	  // nicht verwendete Signale für den 1. Schritt und eventuell weitere Schritte
	  (*#sxSendBuf.sxSTW1.Jog1         := False;
	          #sxSendBuf.sxSTW1.Jog2         := False;
	          #sxSendBuf.sxEPosSTW1.MdiTyp   := False;
	          #sxSendBuf.sxEPosSTW1.MdiPos   := False;
	          #sxSendBuf.sxEPosSTW1.MdiNeg   := False;
	          #sxSendBuf.sxEPosSTW1.MdiSetup := False;
	          #sxSendBuf.sxEPosSTW2.SetRefPt := False;
	          #sxSendBuf.sxEPosSTW2.JogInc   := False;
	          #sxSendBuf.sxEPosSTW2.RefStDi  := False;
	          #sxSendBuf.sxSTW1.RefStart     := False;
	          #sxSendBuf.sxEPosSTW2.RefTyp   := False;
	          #sxSendBuf.sxEPosSTW1.MdiStart := False;*)
	  #sxSendBuf.STW1.%X8 := False;
	  #sxSendBuf.STW1.%X9 := False;
	  #sxSendBuf.EPosSTW1.%X8 := False;
	  #sxSendBuf.EPosSTW1.%X9 := False;
	  #sxSendBuf.EPosSTW1.%X10 := False;
	  #sxSendBuf.EPosSTW1.%X14 := False;
	  #sxSendBuf.EPosSTW2.%X1 := False;
	  #sxSendBuf.EPosSTW2.%X5 := False;
	  #sxSendBuf.EPosSTW2.%X9 := False;
	  #sxSendBuf.STW1.%X11 := False;
	  #sxSendBuf.EPosSTW2.%X8 := False;
	  #sxSendBuf.EPosSTW1.%X15 := False;
	  
	  // Nach dem Einschalten des Antriebes, prüfen ob der Antrieb betriebsbereit, in Operation ohne Fehler und Warnung ist, 
	  // dann die Betriebsart MDI / Sollwertvorgabe Start gesetzt werden
	  IF #sbOff1 AND #sbReady AND #sbIOp AND NOT #sbFault THEN
	    
	    // Betriebsart MDI / Sollwertdirektvorgabe setzen
	    //#sxSendBuf.sxEPosSTW1.MdiStart := True;
	    #sxSendBuf.EPosSTW1.%X15 := True;
	    
	    // Positioniertyp auf absolutes Positionieren stellen 
	    //#sxSendBuf.sxEPosSTW1.MdiTyp := True;
	    #sxSendBuf.EPosSTW1.%X8 := True;
	    
	    // die Richtungswahl für das Positionieren auf positive Richtung oder negative Richtung einstellen
	    IF #Positive AND NOT #Negative THEN
	      
	      // positive Richtung
	      //#sxSendBuf.sxEPosSTW1.MdiPos := True;
	      #sxSendBuf.EPosSTW1.%X9 := True;
	      
	      // negative Richtung
	      //#sxSendBuf.sxEPosSTW1.MdiNeg := False;
	      #sxSendBuf.EPosSTW1.%X10 := False;
	      
	      // die Richtungswahl für das Positionieren auf negative Richtung einstellen                
	    ELSIF NOT #Positive AND #Negative THEN
	      
	      // positive Richtung
	      //#sxSendBuf.sxEPosSTW1.MdiPos := False;
	      #sxSendBuf.EPosSTW1.%X9 := False;
	      
	      // negative Richtung
	      //#sxSendBuf.sxEPosSTW1.MdiNeg := True;
	      #sxSendBuf.EPosSTW1.%X10 := True;
	      
	      // die Richtungswahl für das Positionieren auf keine Richtung einstellen                
	    ELSE
	      
	      // positive Richtung
	      //#sxSendBuf.sxEPosSTW1.MdiPos := False;
	      #sxSendBuf.EPosSTW1.%X9 := False;
	      
	      // negative Richtung
	      //#sxSendBuf.sxEPosSTW1.MdiNeg := False;
	      #sxSendBuf.EPosSTW1.%X10 := False;
	      
	    END_IF;
	    
	    // Nach dem Einschalten des Antriebes und dem Betriebsart MDI / Sollwertvorgabe starten, 
	    // ein Paar Zyklen warten bevor die Flanke für die Sollwertübernahme MDI gesetzt werden kann
	    IF #sbMdiStart AND (#siMdiStartCyc < #siCycWait) THEN
	      #siMdiStartCyc := #siMdiStartCyc + 1;
	    ELSE
	      // Flanke Sollwertübernahme MDI
	      //#sxSendBuf.sxSTW1.TrvStart := #Execute;
	      #sxSendBuf.STW1.%X6 := #sbExecute;
	      
	    END_IF;
	    
	    // "Fliegendes Referentieren" aktivieren
	    // "Fliegendes Referenzieren" erst nach Einschalten des Antriebes möglich
	    IF #sbRefTyp THEN
	      
	      // Referenziertyp auf "Fliegendes Referenzieren" einstellen
	      //#sxSendBuf.sxEPosSTW2.RefTyp := True;
	      #sxSendBuf.EPosSTW2.%X8 := True;
	      
	      // Nach der Anwahl des Referenziertyps "Fliegendes Referenzieren", 
	      // ein Zyklus später kann das Referenzieren gestartet
	      IF (#siRefTypCyc = 0) THEN
	        #siRefTypCyc := #siRefTypCyc + 1;
	      ELSE
	        // Referenzieren starten
	        //#sxSendBuf.sxSTW1.RefStart := True;
	        #sxSendBuf.STW1.%X11 := True;
	        
	      END_IF;
	    END_IF;
	  END_IF;
	  
	  // Betriebsart "Positionieren als Einrichten positiv" oder "Positionieren als Einrichten negativ"
	ELSIF #siModePos = 3 AND #sbModePos THEN
	  
	  // Antrieb einschalten
	  //#sxSendBuf.sxSTW1.Off1 := #sbOff1;
	  #sxSendBuf.STW1.%X0 := #sbOff1;
	  
	  // nicht verwendete Signale für den 1. Schritt und eventuell weitere Schritte
	  (*#sxSendBuf.sxSTW1.Jog1           := False;
	          #sxSendBuf.sxSTW1.Jog2           := False;
	          #sxSendBuf.sxEPosSTW1.MdiTyp     := False;
	          #sxSendBuf.sxEPosSTW1.MdiPos     := False;
	          #sxSendBuf.sxEPosSTW1.MdiNeg     := False;
	          #sxSendBuf.sxEPosSTW1.MdiSetup   := False;
	          #sxSendBuf.sxEPosSTW2.SetRefPt   := False;
	          #sxSendBuf.sxEPosSTW2.JogInc     := False;
	          #sxSendBuf.sxEPosSTW2.RefStDi    := False;
	          #sxSendBuf.sxSTW1.RefStart       := False;
	          #sxSendBuf.sxEPosSTW2.RefTyp     := False;
	          #sxSendBuf.sxEPosSTW1.MdiStart   := False;*)
	  #sxSendBuf.STW1.%X8 := False;
	  #sxSendBuf.STW1.%X9 := False;
	  #sxSendBuf.EPosSTW1.%X8 := False;
	  #sxSendBuf.EPosSTW1.%X9 := False;
	  #sxSendBuf.EPosSTW1.%X10 := False;
	  #sxSendBuf.EPosSTW1.%X14 := False;
	  #sxSendBuf.EPosSTW2.%X1 := False;
	  #sxSendBuf.EPosSTW2.%X5 := False;
	  #sxSendBuf.EPosSTW2.%X9 := False;
	  #sxSendBuf.STW1.%X11 := False;
	  #sxSendBuf.EPosSTW2.%X8 := False;
	  #sxSendBuf.EPosSTW1.%X15 := False;
	  
	  // Nach dem Einschalten des Antriebes, prüfen ob der Antrieb betriebsbereit, in Operation ohne Fehler und Warnung ist, 
	  // dann die Betriebsart MDI / Sollwertvorgabe Start gesetzt werden
	  IF #sbOff1 AND #sbReady AND #sbIOp AND NOT #sbFault THEN
	    
	    // Betriebsart MDI / Sollwertdirektvorgabe setzen
	    //#sxSendBuf.sxEPosSTW1.MdiStart := True;
	    #sxSendBuf.EPosSTW1.%X15 := True;
	    
	    // Positioniertyp auf absolutes Positionieren stellen 
	    //#sxSendBuf.sxEPosSTW1.MdiTyp := True;
	    #sxSendBuf.EPosSTW1.%X8 := True;
	    
	    // die Anwahl für MDI Modus auf Einrichten einstellen
	    //#sxSendBuf.sxEPosSTW1.MdiSetup := True;
	    #sxSendBuf.EPosSTW1.%X14 := True;
	    
	    // die Richtungswahl für das Positionieren auf positive Richtung oder negative Richtung einstellen
	    IF #Positive AND NOT #Negative THEN
	      
	      // positive Richtung
	      //#sxSendBuf.sxEPosSTW1.MdiPos := True;
	      #sxSendBuf.EPosSTW1.%X9 := True;
	      
	      // negative Richtung
	      //#sxSendBuf.sxEPosSTW1.MdiNeg := False;
	      #sxSendBuf.EPosSTW1.%X10 := False;
	      
	      // die Richtungswahl für das Positionieren auf negative Richtung einstellen                
	    ELSIF NOT #Positive AND #Negative THEN
	      
	      // positive Richtung
	      //#sxSendBuf.sxEPosSTW1.MdiPos := False;
	      #sxSendBuf.EPosSTW1.%X9 := False;
	      
	      // negative Richtung
	      //#sxSendBuf.sxEPosSTW1.MdiNeg := True;
	      #sxSendBuf.EPosSTW1.%X10 := True;
	      
	      // die Richtungswahl für das Positionieren auf keine Richtung einstellen                
	    ELSE
	      
	      // positive Richtung
	      //#sxSendBuf.sxEPosSTW1.MdiPos := False;
	      #sxSendBuf.EPosSTW1.%X9 := False;
	      
	      // negative Richtung
	      //#sxSendBuf.sxEPosSTW1.MdiNeg := False;
	      #sxSendBuf.EPosSTW1.%X10 := False;
	      
	    END_IF;
	    
	    // Nach dem Einschalten des Antriebes und dem Betriebsart MDI / Sollwertvorgabe starten, 
	    // ein Paar Zyklen warten bevor die Flanke für die Sollwertübernahme MDI gesetzt werden kann
	    IF #sbMdiStart AND (#siMdiStartCyc < #siCycWait) THEN
	      #siMdiStartCyc := #siMdiStartCyc + 1;
	    ELSE
	      // Flanke Sollwertübernahme MDI
	      //#sxSendBuf.sxSTW1.TrvStart := #Execute;
	      #sxSendBuf.STW1.%X6 := #sbExecute;
	      
	    END_IF;
	    
	    // "Fliegendes Referentieren" aktivieren
	    // "Fliegendes Referenzieren" erst nach Einschalten des Antriebes möglich
	    IF #sbRefTyp THEN
	      
	      // Referenziertyp auf "Fliegendes Referenzieren" einstellen
	      //#sxSendBuf.sxEPosSTW2.RefTyp := True;
	      #sxSendBuf.EPosSTW2.%X8 := True;
	      
	      // Nach der Anwahl des Referenziertyps "Fliegendes Referenzieren", 
	      // ein Zyklus später kann das Referenzieren gestartet
	      IF (#siRefTypCyc = 0) THEN
	        #siRefTypCyc := #siRefTypCyc + 1;
	      ELSE
	        // Referenzieren starten
	        //#sxSendBuf.sxSTW1.RefStart := True;
	        #sxSendBuf.STW1.%X11 := True;
	        
	      END_IF;
	    END_IF;
	  END_IF;
	  
	  // Hauptbetriebsart "Referenzieren" (Reference)
	  // Betriebsart "Referenzieren - Referenzpunktfahrt positiv" oder "Referenzieren - Referenzpunktfahrt negativ"
	ELSIF #siModePos = 4 AND #sbModePos THEN
	  
	  // Antrieb einschalten
	  //#sxSendBuf.sxSTW1.Off1 := #sbOff1;
	  #sxSendBuf.STW1.%X0 := #sbOff1;
	  
	  // nicht verwendete Signale für den 1. Schritt und eventuell weitere Schritte
	  (*#sxSendBuf.sxSTW1.Jog1         := False;
	          #sxSendBuf.sxSTW1.Jog2         := False;
	          #sxSendBuf.sxEPosSTW1.MdiStart := False;
	          #sxSendBuf.sxEPosSTW2.SetRefPt := False;
	          #sxSendBuf.sxEPosSTW2.JogInc   := False;
	          #sxSendBuf.sxEPosSTW2.RefTyp   := False;
	          #sxSendBuf.sxSTW1.RefStart     := False;
	          #sxSendBuf.sxEPosSTW2.RefStDi  := False;*)
	  #sxSendBuf.STW1.%X8 := False;
	  #sxSendBuf.STW1.%X9 := False;
	  #sxSendBuf.EPosSTW1.%X15 := False;
	  #sxSendBuf.EPosSTW2.%X1 := False;
	  #sxSendBuf.EPosSTW2.%X5 := False;
	  #sxSendBuf.EPosSTW2.%X8 := False;
	  #sxSendBuf.STW1.%X11 := False;
	  #sxSendBuf.EPosSTW2.%X9 := False;
	  
	  // Nach dem Einschalten des Antriebes, prüfen ob der Antrieb betriebsbereit, in Operation ohne Fehler und Warnung ist, 
	  // dann die Betriebsart MDI / Sollwertvorgabe Start gesetzt werden
	  IF #sbOff1 AND #sbReady AND #sbIOp AND NOT #sbFault THEN
	    
	    // Referenzieren starten
	    //#sxSendBuf.sxSTW1.RefStart := #Execute;
	    #sxSendBuf.STW1.%X11 := #sbExecute;
	    
	    // die Richtungswahl für das Referenzpunktfahrt positiv einstellen
	    IF #Positive AND NOT #Negative THEN
	      
	      // positive Referenzpunktfahrt
	      //#sxSendBuf.sxEPosSTW2.RefStDi := False;
	      #sxSendBuf.EPosSTW2.%X9 := False;
	      
	      // die Richtungswahl für das Referenzpunktfahrt negativ einstellen                
	    ELSIF NOT #Positive AND #Negative THEN
	      
	      // negative Referenzpunktfahrt
	      //#sxSendBuf.sxEPosSTW2.RefStDi := True;
	      #sxSendBuf.EPosSTW2.%X9 := True;
	      
	    END_IF;
	  END_IF;
	  
	  // Betriebsart "Referenzieren - Referenzpunkt setzen"
	ELSIF #siModePos = 5 AND #sbModePos THEN
	  
	  // Antrieb einschalten
	  //#sxSendBuf.sxSTW1.Off1 := #sbOff1;
	  #sxSendBuf.STW1.%X0 := #sbOff1;
	  
	  // nicht verwendete Signale für den 1. Schritt und eventuell weitere Schritte
	  (*#sxSendBuf.sxSTW1.Jog1          := False;
	          #sxSendBuf.sxSTW1.Jog2          := False;
	          #sxSendBuf.sxSTW1.RefStart      := False;
	          #sxSendBuf.sxEPosSTW1.MdiStart  := False;
	          #sxSendBuf.sxEPosSTW2.JogInc    := False;
	          #sxSendBuf.sxEPosSTW2.RefTyp    := False;
	          #sxSendBuf.sxEPosSTW2.RefStDi   := False;
	          #sxSendBuf.sxEPosSTW2.SetRefPt  := False;*)
	  #sxSendBuf.STW1.%X8 := False;
	  #sxSendBuf.STW1.%X9 := False;
	  #sxSendBuf.STW1.%X11 := False;
	  #sxSendBuf.EPosSTW1.%X15 := False;
	  #sxSendBuf.EPosSTW2.%X5 := False;
	  #sxSendBuf.EPosSTW2.%X8 := False;
	  #sxSendBuf.EPosSTW2.%X9 := False;
	  #sxSendBuf.EPosSTW2.%X1 := False;
	  
	  // Nach dem Einschalten des Antriebes, prüfen ob der Antrieb betriebsbereit, in Operation ohne Fehler und Warnung ist, 
	  // dann die Betriebsart MDI / Sollwertvorgabe Start gesetzt werden
	  IF NOT #sbFault THEN
	    
	    // Referenzpunktfahrt negativ
	    //#sxSendBuf.sxEPosSTW2.SetRefPt := #Execute;
	    #sxSendBuf.EPosSTW2.%X1 := #sbExecute;
	    
	  END_IF;
	  
	  // Hauptbetriebsart "Verfahrsätze" (Traversing Blocks)
	ELSIF #siModePos = 6 AND #sbModePos THEN
	  
	  // Antrieb einschalten
	  //#sxSendBuf.sxSTW1.Off1 := #sbOff1;
	  #sxSendBuf.STW1.%X0 := #sbOff1;
	  
	  // nicht verwendete Signale für den 1. Schritt und eventuell weitere Schritte
	  (*#sxSendBuf.sxSTW1.Jog1          := False;
	          #sxSendBuf.sxSTW1.Jog2          := False;
	          #sxSendBuf.sxEPosSTW1.MdiTyp    := False;
	          #sxSendBuf.sxEPosSTW1.MdiPos    := False;
	          #sxSendBuf.sxEPosSTW1.MdiNeg    := False;
	          #sxSendBuf.sxEPosSTW1.MdiSetup  := False;
	          #sxSendBuf.sxEPosSTW2.SetRefPt  := False;
	          #sxSendBuf.sxEPosSTW2.JogInc    := False;
	          #sxSendBuf.sxEPosSTW2.RefStDi   := False;
	          #sxSendBuf.sxEPosSTW2.RefTyp    := False;
	          #sxSendBuf.sxSTW1.RefStart      := False;
	          #sxSendBuf.sxEPosSTW1.TrvBit0   := False;
	          #sxSendBuf.sxEPosSTW1.TrvBit1   := False;
	          #sxSendBuf.sxEPosSTW1.TrvBit2   := False;
	          #sxSendBuf.sxEPosSTW1.TrvBit3   := False;
	          #sxSendBuf.sxEPosSTW1.TrvBit4   := False;
	          #sxSendBuf.sxEPosSTW1.TrvBit5   := False;
	          #sxSendBuf.sxEPosSTW1.MdiStart  := False;*)
	  #sxSendBuf.STW1.%X8 := False;
	  #sxSendBuf.STW1.%X9 := False;
	  #sxSendBuf.EPosSTW1.%X8 := False;
	  #sxSendBuf.EPosSTW1.%X9 := False;
	  #sxSendBuf.EPosSTW1.%X10 := False;
	  #sxSendBuf.EPosSTW1.%X14 := False;
	  #sxSendBuf.EPosSTW2.%X1 := False;
	  #sxSendBuf.EPosSTW2.%X5 := False;
	  #sxSendBuf.EPosSTW2.%X9 := False;
	  #sxSendBuf.EPosSTW2.%X8 := False;
	  #sxSendBuf.STW1.%X11 := False;
	  #sxSendBuf.EPosSTW1.%X0 := False;
	  #sxSendBuf.EPosSTW1.%X1 := False;
	  #sxSendBuf.EPosSTW1.%X2 := False;
	  #sxSendBuf.EPosSTW1.%X3 := False;
	  #sxSendBuf.EPosSTW1.%X4 := False;
	  #sxSendBuf.EPosSTW1.%X5 := False;
	  #sxSendBuf.EPosSTW1.%X15 := False;
	  
	  // Bei der Auswahl der Verfahrsätze entspricht die Position der Verfahrensatznummer 
	  // Verfahrsatznummer aus der Position ermitteln und in die einzelnen Bit's aufteilen
	  // Es sind die Verfahrsatznummern 0 - 63 möglich
	  IF (DINT_TO_INT(#Position) < 0) OR (DINT_TO_INT(#Position) > 63) THEN
	    // Fehler, ungültiger Verfahrsatznummer
	    #swStatus := 16#8204;
	    #Error := True;
	  ELSE
	    // Fehler wieder zurücknehmen, wenn er mal ausgelöst wurde
	    IF #swStatus = 16#8204 THEN
	      #swStatus := 16#7002;
	      #Error := False;
	    END_IF;
	    
	    // Verfahrsatznummer Bit 0 ermitteln
	    IF (DINT_TO_WORD(#Position) AND W#16#01) = W#16#01 THEN
	      //#sxSendBuf.sxEPosSTW1.TrvBit0 := True;
	      #sxSendBuf.EPosSTW1.%X0 := True;
	    END_IF;
	    
	    // Verfahrsatznummer Bit 1 ermitteln
	    IF (DINT_TO_WORD(#Position) AND W#16#02) = W#16#02 THEN
	      //#sxSendBuf.sxEPosSTW1.TrvBit1 := True;
	      #sxSendBuf.EPosSTW1.%X1 := True;
	    END_IF;
	    
	    // Verfahrsatznummer Bit 2 ermitteln
	    IF (DINT_TO_WORD(#Position) AND W#16#04) = W#16#04 THEN
	      //#sxSendBuf.sxEPosSTW1.TrvBit2 := True;
	      #sxSendBuf.EPosSTW1.%X2 := True;
	    END_IF;
	    
	    // Verfahrsatznummer Bit 3 ermitteln
	    IF (DINT_TO_WORD(#Position) AND W#16#08) = W#16#08 THEN
	      //#sxSendBuf.sxEPosSTW1.TrvBit3 := True;
	      #sxSendBuf.EPosSTW1.%X3 := True;
	    END_IF;
	    
	    // Verfahrsatznummer Bit 4 ermitteln
	    IF (DINT_TO_WORD(#Position) AND W#16#10) = W#16#10 THEN
	      //#sxSendBuf.sxEPosSTW1.TrvBit4 := True;
	      #sxSendBuf.EPosSTW1.%X4 := True;
	    END_IF;
	    
	    // Verfahrsatznummer Bit 5 ermitteln
	    IF (DINT_TO_WORD(#Position) AND W#16#20) = W#16#20 THEN
	      //#sxSendBuf.sxEPosSTW1.TrvBit5 := True;
	      #sxSendBuf.EPosSTW1.%X5 := True;
	    END_IF;
	    
	    // Nach dem Einschalten des Antriebes, prüfen ob der Antrieb betriebsbereit, in Operation ohne Fehler und Warnung ist, 
	    // dann die Betriebsart MDI / Sollwertvorgabe Start gesetzt werden
	    IF #sbOff1 AND #sbReady AND #sbIOp AND NOT #sbFault THEN
	      
	      #sxSendBuf.STW1.%X6 := #sbExecute;
	      
	      // "Fliegendes Referentieren" aktivieren
	      // "Fliegendes Referenzieren" erst nach Einschalten des Antriebes möglich
	      IF #sbRefTyp THEN
	        
	        // Referenziertyp auf "Fliegendes Referenzieren" einstellen
	        //#sxSendBuf.sxEPosSTW2.RefTyp := True;
	        #sxSendBuf.EPosSTW2.%X8 := True;
	        
	        // Nach der Anwahl des Referenziertyps "Fliegendes Referenzieren", 
	        // ein Zyklus später kann das Referenzieren gestartet
	        IF (#siRefTypCyc = 0) THEN
	          #siRefTypCyc := #siRefTypCyc + 1;
	        ELSE
	          // Referenzieren starten
	          //#sxSendBuf.sxSTW1.RefStart := True;
	          #sxSendBuf.STW1.%X11 := True;
	        END_IF;
	      END_IF;
	    END_IF;
	  END_IF;
	  
	  // Hauptbetriebsart "Tippen" (Jogging)
	  // Betriebsart "Tippen positiv" oder "Tippen negativ" angewählt 
	ELSIF #siModePos = 7 AND #sbModePos THEN
	  
	  // Antrieb einschalten
	  //#sxSendBuf.sxSTW1.Off1 := #sbOff1;
	  #sxSendBuf.STW1.%X0 := #sbOff1;
	  
	  // nicht verwendete Signale für den 1. Schritt und eventuell weitere Schritte
	  (*#sxSendBuf.sxEPosSTW1.MdiStart := False;
	          #sxSendBuf.sxEPosSTW2.JogInc   := False;
	          #sxSendBuf.sxSTW1.Jog1         := False;
	          #sxSendBuf.sxSTW1.Jog2         := False;
	          #sxSendBuf.sxEPosSTW2.RefTyp   := False;
	          #sxSendBuf.sxSTW1.RefStart     := False;
	          #sxSendBuf.sxEPosSTW2.SetRefPt  := False;*)
	  
	  #sxSendBuf.EPosSTW1.%X15 := False;
	  #sxSendBuf.EPosSTW2.%X5 := False;
	  #sxSendBuf.STW1.%X8 := False;
	  #sxSendBuf.STW1.%X9 := False;
	  #sxSendBuf.EPosSTW2.%X8 := False;
	  #sxSendBuf.STW1.%X11 := False;
	  #sxSendBuf.EPosSTW2.%X1 := False;
	  
	  // Nach dem Einschalten des Antriebes, prüfen ob der Antrieb betriebsbereit, in Operation ohne Fehler und Warnung ist, 
	  // dann kann Tippen positiv oder negativ gesetzt werden
	  IF #sbOff1 AND #sbReady AND #sbIOp AND NOT #sbFault THEN
	    
	    // Tippen positiv
	    IF #Jog1 AND NOT #Jog2 THEN
	      //#sxSendBuf.sxSTW1.Jog1 := True;
	      #sxSendBuf.STW1.%X8 := True;
	    END_IF;
	    
	    // Tippen negativ
	    IF #Jog2 AND NOT #Jog1 THEN
	      //#sxSendBuf.sxSTW1.Jog2 := True;
	      #sxSendBuf.STW1.%X9 := True;
	    END_IF;
	    
	    // "Fliegendes Referentieren" aktivieren
	    // "Fliegendes Referenzieren" erst nach Einschalten des Antriebes möglich
	    IF #sbRefTyp THEN
	      
	      // Referenziertyp auf "Fliegendes Referenzieren" einstellen
	      //#sxSendBuf.sxEPosSTW2.RefTyp := #FlyRef;
	      #sxSendBuf.EPosSTW2.%X8 := #FlyRef;
	      
	      // Nach der Anwahl des Referenziertyps "Fliegendes Referenzieren", 
	      // ein Zyklus später kann das Referenzieren gestartet
	      IF (#siRefTypCyc = 0) THEN
	        #siRefTypCyc := #siRefTypCyc + 1;
	      ELSE
	        // Referenzieren starten
	        //#sxSendBuf.sxSTW1.RefStart := True;
	        #sxSendBuf.STW1.%X11 := True;
	      END_IF;
	    END_IF;
	  END_IF;
	  
	  // Betriebsart "Tippen positiv / Tippen negativ inkrementell" 
	ELSIF #siModePos = 8 AND #sbModePos THEN
	  
	  // Antrieb einschalten
	  //#sxSendBuf.sxSTW1.OFF1 := #sbOff1;
	  #sxSendBuf.STW1.%X0 := #sbOff1;
	  
	  // nicht verwendete Signale für den 1. Schritt und eventuell weitere Schritte
	  (*#sxSendBuf.sxEPosSTW1.MdiStart := False;
	          #sxSendBuf.sxEPosSTW2.JogInc   := False;
	          #sxSendBuf.sxSTW1.Jog1         := False;
	          #sxSendBuf.sxSTW1.Jog2         := False;
	          #sxSendBuf.sxSTW1.RefStart     := False;
	          #sxSendBuf.sxEPosSTW2.RefTyp   := False;
	          #sxSendBuf.sxEPosSTW2.SetRefPt  := False;*)
	  
	  #sxSendBuf.EPosSTW1.%X15 := False;
	  #sxSendBuf.EPosSTW2.%X5 := False;
	  #sxSendBuf.STW1.%X8 := False;
	  #sxSendBuf.STW1.%X9 := False;
	  #sxSendBuf.STW1.%X11 := False;
	  #sxSendBuf.EPosSTW2.%X8 := False;
	  #sxSendBuf.EPosSTW2.%X1 := False;
	  
	  // Nach dem Einschalten des Antriebes, ein Paar Zyklen warten bevor Tippen negativ gesetzt werden kann
	  // Nach dem Einschalten des Antriebes, prüfen ob der Antrieb betriebsbereit, in Operation ohne Fehler und Warnung ist, 
	  // dann kann Tippen positiv oder negativ gesetzt werden
	  IF #sbOff1 AND #sbReady AND #sbIOp AND NOT #sbFault THEN
	    
	    // Tippen inkrementell einstellen
	    //#sxSendBuf.sxEPosSTW2.JogInc := True;
	    #sxSendBuf.EPosSTW2.%X5 := True;
	    
	    #sbJogInc := True;
	    
	    // Nach dem Einstellen des Antriebes, ein Paar Zyklen warten bevor Tippen negativ oder Tippen positiv gesetz werden kann
	    IF #sbJogInc AND (#siJogIncCyc = 0) THEN
	      #siJogIncCyc := #siJogIncCyc + 1;
	    ELSE
	      
	      // Tippen positiv oder negativ inkrementell zulassen
	      IF #Jog1 XOR #Jog2 THEN
	        
	        //#sxSendBuf.sxSTW1.Jog1 := #Jog1;
	        //#sxSendBuf.sxSTW1.Jog2 := #Jog2;
	        #sxSendBuf.STW1.%X8 := #Jog1;
	        #sxSendBuf.STW1.%X9 := #Jog2;
	      END_IF;
	    END_IF;
	    
	    // "Fliegendes Referentieren" aktivieren
	    // "Fliegendes Referenzieren" erst nach Einschalten des Antriebes möglich
	    IF #sbRefTyp THEN
	      
	      // Referenziertyp auf "Fliegendes Referenzieren" einstellen
	      //#sxSendBuf.sxEPosSTW2.RefTyp := True;
	      #sxSendBuf.EPosSTW2.%X8 := True;
	      
	      // Nach der Anwahl des Referenziertyps "Fliegendes Referenzieren", 
	      // ein Zyklus später kann das Referenzieren gestartet
	      IF (#siRefTypCyc = 0) THEN
	        #siRefTypCyc := #siRefTypCyc + 1;
	      ELSE
	        // Referenzieren starten
	        //#sxSendBuf.sxSTW1.RefStart := True;
	        #sxSendBuf.STW1.%X11 := True;
	      END_IF;
	    END_IF;
	  END_IF;
	ELSE
	  // Werte wieder zurücknehmen
	  (*#sxSendBuf.sxSTW1.Off1          := #Off1;
	          #sxSendBuf.sxSTW1.RejTrvTsk     := False;
	          #sxSendBuf.sxSTW1.TrvStart      := False;
	          #sxSendBuf.sxEPosSTW1.MdiStart  := False;
	          #sxSendBuf.sxSTW1.Jog1          := False;
	          #sxSendBuf.sxSTW1.Jog2          := False;
	          #sxSendBuf.sxEPosSTW1.MdiTyp    := False;
	          #sxSendBuf.sxEPosSTW1.MdiPos    := False;
	          #sxSendBuf.sxEPosSTW1.MdiNeg    := False;
	          #sxSendBuf.sxEPosSTW1.MdiTrTyp  := False;
	          #sxSendBuf.sxEPosSTW1.MdiSetup  := False;
	          #sxSendBuf.sxEPosSTW2.SetRefPt  := False;
	          #sxSendBuf.sxEPosSTW2.RefTyp    := False;
	          #sxSendBuf.sxEPosSTW2.RefStDi   := False;
	          #sxSendBuf.sxEPosSTW2.JogInc    := False;
	          #sxSendBuf.sxSTW1.RefStart      := False;*)
	  
	  #sxSendBuf.STW1.%X0 := #EnableAxis;
	  #sxSendBuf.STW1.%X4 := False;
	  #sxSendBuf.STW1.%X6 := False;
	  #sxSendBuf.EPosSTW1.%X15 := False;
	  #sxSendBuf.STW1.%X8 := False;
	  #sxSendBuf.STW1.%X9 := False;
	  #sxSendBuf.EPosSTW1.%X8 := False;
	  #sxSendBuf.EPosSTW1.%X9 := False;
	  #sxSendBuf.EPosSTW1.%X10 := False;
	  #sxSendBuf.EPosSTW1.%X12 := False;
	  #sxSendBuf.EPosSTW1.%X14 := False;
	  #sxSendBuf.EPosSTW2.%X1 := False;
	  #sxSendBuf.EPosSTW2.%X8 := False;
	  #sxSendBuf.EPosSTW2.%X9 := False;
	  #sxSendBuf.EPosSTW2.%X5 := False;
	  #sxSendBuf.STW1.%X11 := False;
	END_IF; // Hauptbetriebsart "Verfahrsätze" (Traversing Blocks)
	
	//Den Eingang ConfigEPos auf die einzelnen Bits im Telegramm verschalten
	#sxSendBuf.STW1.%X1 := #ConfigEPos.%X0;
	#sxSendBuf.STW1.%X2 := #ConfigEPos.%X1;
	#sxSendBuf.EPosSTW2.%X14 := #ConfigEPos.%X2;
	#sxSendBuf.EPosSTW2.%X15 := #ConfigEPos.%X3;
	#sxSendBuf.EPosSTW2.%X11 := #ConfigEPos.%X4;
	#sxSendBuf.EPosSTW2.%X10 := #ConfigEPos.%X5;
	#sxSendBuf.EPosSTW2.%X2 := #ConfigEPos.%X6;
	#sxSendBuf.STW1.%X13 := #ConfigEPos.%X7;
	#sxSendBuf.EPosSTW1.%X12 := #ConfigEPos.%X8;
	#sxSendBuf.STW2.%X0 := #ConfigEPos.%X9;
	#sxSendBuf.STW2.%X1 := #ConfigEPos.%X10;
	#sxSendBuf.STW2.%X2 := #ConfigEPos.%X11;
	#sxSendBuf.STW2.%X3 := #ConfigEPos.%X12;
	#sxSendBuf.STW2.%X4 := #ConfigEPos.%X13;
	#sxSendBuf.STW2.%X7 := #ConfigEPos.%X14;
	#sxSendBuf.STW1.%X12 := #ConfigEPos.%X15;
	#sxSendBuf.STW1.%X14 := #ConfigEPos.%X16;
	#sxSendBuf.STW1.%X15 := #ConfigEPos.%X17;
	#sxSendBuf.EPosSTW1.%X6 := #ConfigEPos.%X18;
	#sxSendBuf.EPosSTW1.%X7 := #ConfigEPos.%X19;
	#sxSendBuf.EPosSTW1.%X11 := #ConfigEPos.%X20;
	#sxSendBuf.EPosSTW1.%X13 := #ConfigEPos.%X21;
	#sxSendBuf.EPosSTW2.%X3 := #ConfigEPos.%X22;
	#sxSendBuf.EPosSTW2.%X4 := #ConfigEPos.%X23;
	#sxSendBuf.EPosSTW2.%X6 := #ConfigEPos.%X24;
	#sxSendBuf.EPosSTW2.%X7 := #ConfigEPos.%X25;
	#sxSendBuf.EPosSTW2.%X12 := #ConfigEPos.%X26;
	#sxSendBuf.EPosSTW2.%X13 := #ConfigEPos.%X27;
	#sxSendBuf.STW2.%X5 := #ConfigEPos.%X28;
	#sxSendBuf.STW2.%X6 := #ConfigEPos.%X29;
	#sxSendBuf.STW2.%X8 := #ConfigEPos.%X30;
	#sxSendBuf.STW2.%X9 := #ConfigEPos.%X31;
	
	
	#swSendBuf[0] := #sxSendBuf.STW1;
	#swSendBuf[1] := #sxSendBuf.EPosSTW1;
	#swSendBuf[2] := #sxSendBuf.EPosSTW2;
	#swSendBuf[3] := #sxSendBuf.STW2;
	#swSendBuf[4] := #sxSendBuf.OverrideV;
	#swSendBuf[5] := #sxSendBuf.Position.%W1;
	#swSendBuf[6] := #sxSendBuf.Position.%W0;
	#swSendBuf[7] := #sxSendBuf.Velocity.%W1;
	#swSendBuf[8] := #sxSendBuf.Velocity.%W0;
	#swSendBuf[9] := #sxSendBuf.OverrideA;
	#swSendBuf[10] := #sxSendBuf.OverrideD;
	#swSendBuf[11] := #sxSendBuf.Reserve;
	
	//Prozessdaten zur Signalbaugruppe schreiben
	#piRetSFC := DPWR_DAT(LADDR := #HWIDSTW,
	                      RECORD := #swSendBuf);
	
	// Fehler der Rückmeldung ausgeben
	#DiagID := INT_TO_WORD(#piRetSFC);
	
	//kein Fehler beim Schreiben
	IF #piRetSFC = 0 THEN
	  
	  // Fehler wieder zurück nehmen
	  IF (#swStatus = 16#8601) THEN
	    #swStatus := 16#7002;
	    #Error := False;
	  END_IF;
	  
	  //Prozessdaten von der Signalbaugruppe lesen
	  #piRetSFC := DPRD_DAT(LADDR := #HWIDZSW,
	                        RECORD => #swRecvBuf);
	  
	  // Fehlermeldung der Rückmeldung ausgeben
	  #DiagID := INT_TO_WORD(#piRetSFC);
	  
	  //Fehler beim Lesen (Profibus-Kommunikation unterbrochen)
	  IF #piRetSFC <> 0 THEN
	    
	    // Fehler
	    #Error := TRUE;
	    #swStatus := 16#8600;
	    
	    // Zustandsworte löschen
	    #sxRecvBuf.ZSW1 := W#16#0;
	    #sxRecvBuf.EPosZSW1 := W#16#0;
	    #sxRecvBuf.EPosZSW2 := W#16#0;
	    #sxRecvBuf.ZSW2 := W#16#0;
	    #sxRecvBuf.NotUsed := W#16#00;
	    #sxRecvBuf.Position := DW#16#00;
	    #sxRecvBuf.Velocity := DW#16#00;
	    #sxRecvBuf.ErrNr := W#16#00;
	    #sxRecvBuf.WarnNr := W#16#00;
	    #sxRecvBuf.Reserve := W#16#00;
	    
	    // Werte auslesen
	  ELSE
	    
	    // Fehler wieder zurück nehmen
	    IF (#swStatus = 16#8600) THEN
	      #swStatus := 16#7002;
	      #Error := False;
	    END_IF;
	    
	    #sxRecvBuf.ZSW1 := #swRecvBuf[0];
	    #sxRecvBuf.EPosZSW1 := #swRecvBuf[1];
	    #sxRecvBuf.EPosZSW2 := #swRecvBuf[2];
	    #sxRecvBuf.ZSW2 := #swRecvBuf[3];
	    #sxRecvBuf.NotUsed := #swRecvBuf[4];
	    #sxRecvBuf.Position.%W1 := #swRecvBuf[5];
	    #sxRecvBuf.Position.%W0 := #swRecvBuf[6];
	    #sxRecvBuf.Velocity.%W1 := #swRecvBuf[7];
	    #sxRecvBuf.Velocity.%W0 := #swRecvBuf[8];
	    #sxRecvBuf.ErrNr := #swRecvBuf[9];
	    #sxRecvBuf.WarnNr := #swRecvBuf[10];
	    #sxRecvBuf.Reserve := #swRecvBuf[11];
	    
	    // ZSW1 aufbereiten
	    //#Busy := #sxRecvBuf.sxZSW1.IOp;
	    #sbBusy := #sxRecvBuf.ZSW1.%X2;
	    
	    // Fehler auswerten
	    IF #sxRecvBuf.ZSW1.%X3 THEN
	      #swStatus := 16#8401;
	      #Error := True;
	    ELSIF #sxRecvBuf.ZSW1.%X6 THEN
	      #swStatus := 16#8402;
	      #Error := True;
	    ELSE
	      // Fehler wieder zurück nehmen
	      IF (#swStatus = 16#8401) OR (#swStatus = 16#8402) THEN
	        #swStatus := 16#7002;
	        #Error := False;
	      END_IF;
	    END_IF;
	    
	    // EPOS_ZSW1            
	    // EPOS-Wort-1 BIT 00 --> 1 = Active traversing block bit 0
	    //IF #sxRecvBuf.sxEPosZSW1.ActTrvBit0 THEN
	    IF #sxRecvBuf.EPosZSW1.%X0 THEN
	      #swEPosZSW1 := #swEPosZSW1 OR W#16#01;
	    ELSE
	      #swEPosZSW1 := #swEPosZSW1 AND W#16#FFFE;
	    END_IF;
	    
	    // EPOS-Wort-1 Bit 01 --> 1 = Active traversing block bit 1
	    //IF #sxRecvBuf.sxEPosZSW1.ActTrvBit1 THEN
	    IF #sxRecvBuf.EPosZSW1.%X1 THEN
	      #swEPosZSW1 := #swEPosZSW1 OR W#16#02;
	    ELSE
	      #swEPosZSW1 := #swEPosZSW1 AND W#16#FFFD;
	    END_IF;
	    
	    // EPOS-Wort-1 Bit 02 --> 1 = Active traversing block bit 2
	    //IF #sxRecvBuf.sxEPosZSW1.ActTrvBit2 THEN
	    IF #sxRecvBuf.EPosZSW1.%X2 THEN
	      #swEPosZSW1 := #swEPosZSW1 OR W#16#04;
	    ELSE
	      #swEPosZSW1 := #swEPosZSW1 AND W#16#FFFB;
	    END_IF;
	    
	    // EPOS-Wort-1 Bit 03 --> 1 = Active traversing block bit 3
	    //IF #sxRecvBuf.sxEPosZSW1.ActTrvBit3 THEN
	    IF #sxRecvBuf.EPosZSW1.%X3 THEN
	      #swEPosZSW1 := #swEPosZSW1 OR W#16#08;
	    ELSE
	      #swEPosZSW1 := #swEPosZSW1 AND W#16#FFF7;
	    END_IF;
	    
	    // EPOS-Wort-1 Bit 04 --> 1 = Active traversing block bit 4 
	    //IF #sxRecvBuf.sxEPosZSW1.ActTrvBit4 THEN
	    IF #sxRecvBuf.EPosZSW1.%X4 THEN
	      #swEPosZSW1 := #swEPosZSW1 OR W#16#10;
	    ELSE
	      #swEPosZSW1 := #swEPosZSW1 AND W#16#FFEF;
	    END_IF;
	    
	    // EPOS-Wort-1 Bit 05 --> 1 = Active traversing block bit 5
	    //IF #sxRecvBuf.sxEPosZSW1.ActTrvBit5 THEN
	    IF #sxRecvBuf.EPosZSW1.%X5 THEN
	      #swEPosZSW1 := #swEPosZSW1 OR W#16#20;
	    ELSE
	      #swEPosZSW1 := #swEPosZSW1 AND W#16#FFDF;
	    END_IF;
	    
	    // EPOS-Wort-1 Bit 08 --> 1 = STOP cam minus active
	    //IF #sxRecvBuf.sxEPosZSW1.StpCamMinAct THEN
	    IF #sxRecvBuf.EPosZSW1.%X8 THEN
	      #swEPosZSW1 := #swEPosZSW1 OR W#16#100;
	    ELSE
	      #swEPosZSW1 := #swEPosZSW1 AND W#16#FEFF;
	    END_IF;
	    
	    // EPOS-Wort-1 Bit 09 --> 1 = STOP cam plus active
	    //IF #sxRecvBuf.sxEPosZSW1.StpCamPlsAct THEN
	    IF #sxRecvBuf.EPosZSW1.%X9 THEN
	      #swEPosZSW1 := #swEPosZSW1 OR W#16#200;
	    ELSE
	      #swEPosZSW1 := #swEPosZSW1 AND W#16#FDFF;
	    END_IF;
	    
	    // EPOS-Wort-1 Bit 10 --> 1 = Jogging active
	    //IF #sxRecvBuf.sxEPosZSW1.JogAct THEN
	    IF #sxRecvBuf.EPosZSW1.%X10 THEN
	      #swEPosZSW1 := #swEPosZSW1 OR W#16#400;
	    ELSE
	      #swEPosZSW1 := #swEPosZSW1 AND W#16#FBFF;
	    END_IF;
	    
	    // EPOS-Wort-1 Bit 11 --> 1 = Reference point approach active
	    //IF #sxRecvBuf.sxEPosZSW1.RefAct THEN
	    IF #sxRecvBuf.EPosZSW1.%X11 THEN
	      #swEPosZSW1 := #swEPosZSW1 OR W#16#800;
	    ELSE
	      #swEPosZSW1 := #swEPosZSW1 AND W#16#F7FF;
	    END_IF;
	    
	    // Anstossen des fliegenden Referenzieren prüfen, wenn die Rückmeldung fehlt dann wiederholen
	    //IF NOT #sxRecvBuf.sxEPosZSW1.FlyRefAct AND #sbRefTyp AND #sxSendBuf.sxSTW1.RefStart THEN
	    IF NOT #sxRecvBuf.EPosZSW1.%X12 AND #sbRefTyp AND #sxSendBuf.STW1.%X11 THEN
	      
	      // Wiederholung anstossen 
	      IF #siRefActRetry < #siRetryMax THEN
	        #siRefActRetry := #siRefActRetry + 1;
	        
	        // Referenzieren starten wieder wegnehmen
	        //#sxSendBuf.sxSTW1.RefStart := False;
	        #sxSendBuf.STW1.%X11 := False;
	      ELSE
	        
	        // Fehlermeldung
	        #swStatus := 16#8403;
	        #Error := True;
	      END_IF;
	    ELSE
	      
	      // Fehler wieder zurücknehmen, wenn er mal ausgelöst wurde
	      IF #swStatus = 16#8403 THEN
	        #swStatus := 16#7002;
	        #Error := False;
	      END_IF;
	      // Zähler zurücksetzen bei Rückmeldung fliegendes Referenzieren jetzt aktiviert oder bei Abwahl der Funktion
	      IF (#sxRecvBuf.EPosZSW1.%X12 AND #sbRefTyp AND #sxSendBuf.STW1.%X11) OR NOT #FlyRef THEN
	        #siRefActRetry := 0;
	      END_IF;
	    END_IF;
	    
	    // EPOS-Wort-1 Bit 12 --> 1 = Flying referencing active
	    //IF #sxRecvBuf.sxEPosZSW1.FlyRefAct THEN
	    IF #sxRecvBuf.EPosZSW1.%X12 THEN
	      #swEPosZSW1 := #swEPosZSW1 OR W#16#1000;
	    ELSE
	      #swEPosZSW1 := #swEPosZSW1 AND W#16#EFFF;
	    END_IF;
	    
	    // EPOS-Wort-1 Bit 13 --> 1 = Traversing block active
	    //IF #sxRecvBuf.sxEPosZSW1.TrvBlAct THEN
	    IF #sxRecvBuf.EPosZSW1.%X13 THEN
	      #swEPosZSW1 := #swEPosZSW1 OR W#16#2000;
	    ELSE
	      #swEPosZSW1 := #swEPosZSW1 AND W#16#DFFF;
	    END_IF;
	    
	    // EPOS-Wort-1 Bit 14 --> 1 = MDI setup active
	    //IF #sxRecvBuf.sxEPosZSW1.MdiStupAct THEN
	    IF #sxRecvBuf.EPosZSW1.%X14 THEN
	      #swEPosZSW1 := #swEPosZSW1 OR W#16#4000;
	    ELSE
	      #swEPosZSW1 := #swEPosZSW1 AND W#16#BFFF;
	    END_IF;
	    
	    // EPOS-Wort-1 Bit 15 --> 1 = MDI positing active
	    //IF #sxRecvBuf.sxEPosZSW1.MdiPosAct THEN
	    IF #sxRecvBuf.EPosZSW1.%X15 THEN
	      #swEPosZSW1 := #swEPosZSW1 OR W#16#8000;
	    ELSE
	      #swEPosZSW1 := #swEPosZSW1 AND W#16#7FFF;
	    END_IF;
	    
	    // EPOS_ZSW2 
	    // EPOS-Wort-2 Bit 00 --> 1 = Tracking mode active
	    //IF #sxRecvBuf.sxEPosZSW2.TrkModeAct THEN
	    IF #sxRecvBuf.EPosZSW2.%X0 THEN
	      #swEPosZSW2 := #swEPosZSW2 OR W#16#01;
	    ELSE
	      #swEPosZSW2 := #swEPosZSW2 AND W#16#FFFE;
	    END_IF;
	    
	    // EPOS-Wort-2 Bit 01 --> 1 = Velocity limit active
	    //IF #sxRecvBuf.sxEPosZSW2.VeloLimAct THEN
	    IF #sxRecvBuf.EPosZSW2.%X1 THEN
	      #swEPosZSW2 := #swEPosZSW2 OR W#16#02;
	    ELSE
	      #swEPosZSW2 := #swEPosZSW2 AND W#16#FFFD;
	    END_IF;
	    
	    // EPOS-Wort-2 Bit 02 --> 1 = Setpoint static
	    //IF #sxRecvBuf.sxEPosZSW2.SetPStat THEN
	    IF #sxRecvBuf.EPosZSW2.%X2 THEN
	      #swEPosZSW2 := #swEPosZSW2 OR W#16#04;
	    ELSE
	      #swEPosZSW2 := #swEPosZSW2 AND W#16#FFFB;
	    END_IF;
	    
	    // EPOS-Wort-2 Bit 03 --> 1 = Printmark outside outer window
	    //IF #sxRecvBuf.sxEPosZSW2.PrnMrkOut THEN
	    IF #sxRecvBuf.EPosZSW2.%X3 THEN
	      #swEPosZSW2 := #swEPosZSW2 OR W#16#08;
	    ELSE
	      #swEPosZSW2 := #swEPosZSW2 AND W#16#FFF7;
	    END_IF;
	    
	    // EPOS-Wort-2 Bit 04 --> 1 = Axis forwards
	    //IF #sxRecvBuf.sxEPosZSW2.FWD THEN
	    IF #sxRecvBuf.EPosZSW2.%X4 THEN
	      #swEPosZSW2 := #swEPosZSW2 OR W#16#10;
	    ELSE
	      #swEPosZSW2 := #swEPosZSW2 AND W#16#FFEF;
	    END_IF;
	    
	    // EPOS-Wort-2 Bit 05 --> 1 = Axis backwards
	    //IF #sxRecvBuf.sxEPosZSW2.BWD THEN
	    IF #sxRecvBuf.EPosZSW2.%X5 THEN
	      #swEPosZSW2 := #swEPosZSW2 OR W#16#20;
	    ELSE
	      #swEPosZSW2 := #swEPosZSW2 AND W#16#FFDF;
	    END_IF;
	    
	    // EPOS-Wort-2 Bit 06 --> 1 = Software limit switch minus active
	    //IF #sxRecvBuf.sxEPosZSW2.SftSwMinAct THEN
	    IF #sxRecvBuf.EPosZSW2.%X6 THEN
	      #swEPosZSW2 := #swEPosZSW2 OR W#16#40;
	    ELSE
	      #swEPosZSW2 := #swEPosZSW2 AND W#16#FFBF;
	    END_IF;
	    
	    // EPOS-Wort-2 Bit 07 --> 1 = Software limit switch plus active
	    //IF #sxRecvBuf.sxEPosZSW2.SftSwPlsAct THEN
	    IF #sxRecvBuf.EPosZSW2.%X7 THEN
	      #swEPosZSW2 := #swEPosZSW2 OR W#16#80;
	    ELSE
	      #swEPosZSW2 := #swEPosZSW2 AND W#16#FF7F;
	    END_IF;
	    
	    // EPOS-Wort-2 Bit 08 --> 1 = Position actual value <= cam position 1
	    //IF #sxRecvBuf.sxEPosZSW2.PosSmCam1 THEN
	    IF #sxRecvBuf.EPosZSW2.%X8 THEN
	      #swEPosZSW2 := #swEPosZSW2 OR W#16#100;
	    ELSE
	      #swEPosZSW2 := #swEPosZSW2 AND W#16#FEFF;
	    END_IF;
	    
	    // EPOS-Wort-2 Bit 09 --> 1 = Position actual value <= cam position 2
	    //IF #sxRecvBuf.sxEPosZSW2.PosSmCam2 THEN
	    IF #sxRecvBuf.EPosZSW2.%X9 THEN
	      #swEPosZSW2 := #swEPosZSW2 OR W#16#200;
	    ELSE
	      #swEPosZSW2 := #swEPosZSW2 AND W#16#FDFF;
	    END_IF;
	    
	    // EPOS-Wort-2 Bit 10 --> 1 = Direct output 1 via traversing block
	    //IF #sxRecvBuf.sxEPosZSW2.TrvOut1 THEN
	    IF #sxRecvBuf.EPosZSW2.%X10 THEN
	      #swEPosZSW2 := #swEPosZSW2 OR W#16#400;
	    ELSE
	      #swEPosZSW2 := #swEPosZSW2 AND W#16#FBFF;
	    END_IF;
	    
	    // EPOS-Wort-2 Bit 11 --> 1 = Direct output 2 via traversing block
	    //IF #sxRecvBuf.sxEPosZSW2.TrvOut2 THEN
	    IF #sxRecvBuf.EPosZSW2.%X11 THEN
	      #swEPosZSW2 := #swEPosZSW2 OR W#16#800;
	    ELSE
	      #swEPosZSW2 := #swEPosZSW2 AND W#16#F7FF;
	    END_IF;
	    
	    // EPOS-Wort-2 Bit 12 --> 1 = Fixed STOP reached
	    //IF #sxRecvBuf.sxEPosZSW2.FxStpRd THEN
	    IF #sxRecvBuf.EPosZSW2.%X12 THEN
	      #swEPosZSW2 := #swEPosZSW2 OR W#16#1000;
	    ELSE
	      #swEPosZSW2 := #swEPosZSW2 AND W#16#EFFF;
	    END_IF;
	    
	    // EPOS-Wort-2 Bit 13 --> 1 = Fixed STOP clamping torque reached
	    //IF #sxRecvBuf.sxEPosZSW2.FxStpTrRd THEN
	    IF #sxRecvBuf.EPosZSW2.%X13 THEN
	      #swEPosZSW2 := #swEPosZSW2 OR W#16#2000;
	    ELSE
	      #swEPosZSW2 := #swEPosZSW2 AND W#16#DFFF;
	    END_IF;
	    
	    // EPOS-Wort-2 Bit 14 --> 1 = Traversing fixed STOP active
	    //IF #sxRecvBuf.sxEPosZSW2.TrvFxStpAct THEN
	    IF #sxRecvBuf.EPosZSW2.%X14 THEN
	      #swEPosZSW2 := #swEPosZSW2 OR W#16#4000;
	    ELSE
	      #swEPosZSW2 := #swEPosZSW2 AND W#16#BFFF;
	    END_IF;
	    
	    // EPOS-Wort-2 Bit 15 --> 1 = Traversing command active
	    //IF #sxRecvBuf.sxEPosZSW2.CmdAct THEN
	    IF #sxRecvBuf.EPosZSW2.%X15 THEN
	      #swEPosZSW2 := #swEPosZSW2 OR W#16#8000;
	    ELSE
	      #swEPosZSW2 := #swEPosZSW2 AND W#16#7FFF;
	    END_IF;
	    
	    #sbReady := #sxRecvBuf.ZSW1.%X1;
	    
	    #AxisEnabled := #sxRecvBuf.ZSW1.%X2;
	    #sbIOp := #sxRecvBuf.ZSW1.%X2;
	    
	    #AxisError := #sxRecvBuf.ZSW1.%X3;
	    #sbFault := #sxRecvBuf.ZSW1.%X3;
	    
	    #AxisWarn := #sxRecvBuf.ZSW1.%X7;
	    #sbAlarm := #sxRecvBuf.ZSW1.%X7;
	    
	    #AxisPosOk := #sxRecvBuf.ZSW1.%X10;
	    #AxisRef := #sxRecvBuf.ZSW1.%X11;
	    #AxisSpFixed := #sxRecvBuf.ZSW1.%X13;
	    
	    #sbAccel := #sxRecvBuf.ZSW1.%X14;
	    #sbDecel := #sxRecvBuf.ZSW1.%X15;
	    
	    #ActVelocity := DWORD_TO_DINT(#sxRecvBuf.Velocity);
	    #ActPosition := DWORD_TO_DINT(#sxRecvBuf.Position);
	    #ActMode := #ModePos;
	    #ActWarn := #sxRecvBuf.WarnNr;
	    #ActFault := #sxRecvBuf.ErrNr;
	    
	    #Lockout := #sxRecvBuf.ZSW1.%X6;
	  END_IF;
	ELSE
	  
	  // Fehler
	  #Error := TRUE;
	  #swStatus := 16#8601;
	  
	END_IF;
	
	// Initialisierung von Ausg㭧en
	#Status := #swStatus;
	#EPosZSW1 := #swEPosZSW1;
	#EPosZSW2 := #swEPosZSW2;
	
END_FUNCTION_BLOCK

FUNCTION_BLOCK "Obj_St2_FB"   // FB200, FBD
{ S7_Optimized_Access := 'TRUE' }
VERSION : 0.1
// stored: AutoNumber false, IsIECCheckEnabled false, IsRetainMemResEnabled false, MemoryReserve 100, SetENOAutomatically false, UDAEnableTagReadback false
   VAR
      Axe_X1 : Struct
         _ActPos : Real;
         _ActVel : Real;
         _Mode : Int;
         Home : Bool;
         Halt : Bool;
         Jog : Bool;
         MoveAbs : Bool;
         MoveRel : Bool;
         MoveVel : Bool;
         PowerOff : Bool;
         PowerOn : Bool;
         SensPos : Bool;
         SensNeg : Bool;
         xBusy : Bool;
         xHomed : Bool;
         xMoveAbsDone : Bool;
         xMoveRelDone : Bool;
         xPower : Bool;
      END_STRUCT;
      Axe_X2 : Struct
         _ActPos : Real;
         _ActVel : Real;
         _Mode : Int;
         Home : Bool;
         Halt : Bool;
         Jog : Bool;
         MoveAbs : Bool;
         MoveRel : Bool;
         MoveVel : Bool;
         PowerOff : Bool;
         PowerOn : Bool;
         SensPos : Bool;
         SensNeg : Bool;
         xBusy : Bool;
         xHomed : Bool;
         xMoveAbsDone : Bool;
         xMoveRelDone : Bool;
         xPower : Bool;
      END_STRUCT;
      Prehenseur_Z : Struct
         _ActPos : Real;
         _ActVel : Real;
         _Mode : Int;
         Home : Bool;
         Halt : Bool;
         Jog : Bool;
         MoveAbs : Bool;
         MoveRel : Bool;
         MoveVel : Bool;
         PowerOff : Bool;
         PowerOn : Bool;
         SensPos : Bool;
         SensNeg : Bool;
         xBusy : Bool;
         xHomed : Bool;
         xMoveAbsDone : Bool;
         xMoveRelDone : Bool;
         xPower : Bool;
      END_STRUCT;
   END_VAR
BEGIN

REGION Network 1: Station 2 - Axe X1
   // //___ ModePose : 
   //          1 ---> Relative positioning
   //          2 ---> Absolute positioning
   //          3 ---> Not supported
   //          4 ---> Referencing - referencing point approach
   //          5 ---> Referencing - set referencing point
   //          6 ---> Traversing block (record mode)
   //          7 ---> Jog
   //          8 ---> Not supported
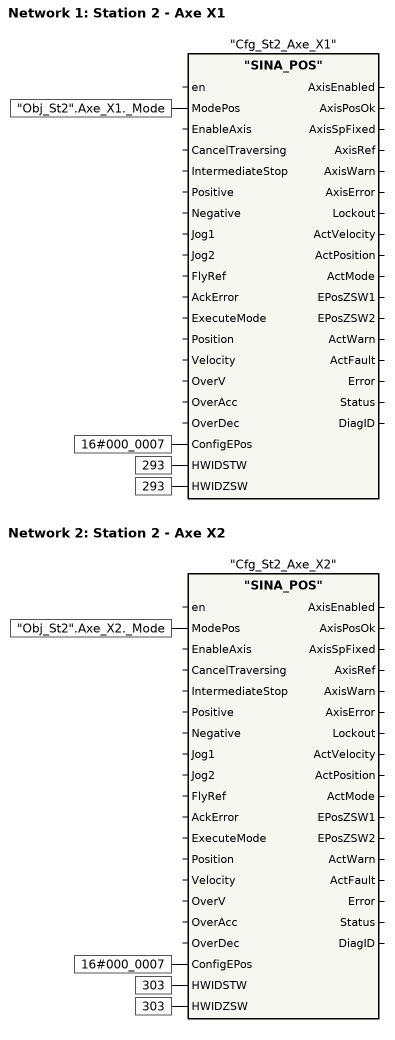
   "Cfg_St2_Axe_X1"(ModePos := "Obj_St2".Axe_X1._Mode,   // "SINA_POS"
                    ConfigEPos := 16#000_0007,
                    HWIDSTW := 293,
                    HWIDZSW := 293);
END_REGION

REGION Network 2: Station 2 - Axe X2
   // //___ ModePose : 
   //          1 ---> Relative positioning
   //          2 ---> Absolute positioning
   //          3 ---> Not supported
   //          4 ---> Referencing - referencing point approach
   //          5 ---> Referencing - set referencing point
   //          6 ---> Traversing block (record mode)
   //          7 ---> Jog
   //          8 ---> Not supported
   "Cfg_St2_Axe_X2"(ModePos := "Obj_St2".Axe_X2._Mode,   // "SINA_POS"
                    ConfigEPos := 16#000_0007,
                    HWIDSTW := 303,
                    HWIDZSW := 303);
END_REGION

REGION Network 3: Station 2 - Prehenseur Z
   // //___ ModePose : 
   //          1 ---> Relative positioning
   //          2 ---> Absolute positioning
   //          3 ---> Not supported
   //          4 ---> Referencing - referencing point approach
   //          5 ---> Referencing - set referencing point
   //          6 ---> Traversing block (record mode)
   //          7 ---> Jog
   //          8 ---> Not supported
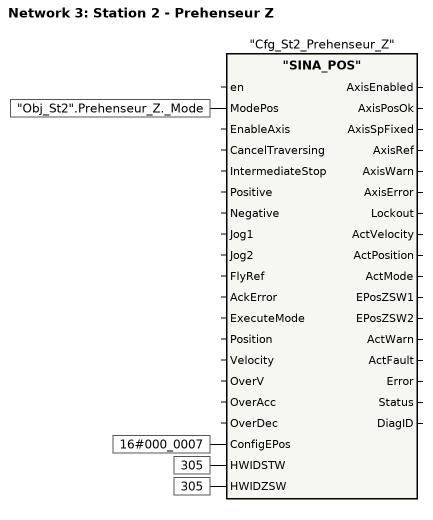
   "Cfg_St2_Prehenseur_Z"(ModePos := "Obj_St2".Prehenseur_Z._Mode,   // "SINA_POS"
                          ConfigEPos := 16#000_0007,
                          HWIDSTW := 305,
                          HWIDZSW := 305);
END_REGION
END_FUNCTION_BLOCK

FUNCTION_BLOCK "Obj_St3_FB"   // FB300, FBD
{ S7_Optimized_Access := 'TRUE' }
VERSION : 0.1
// stored: AutoNumber false, IsIECCheckEnabled false, IsRetainMemResEnabled false, MemoryReserve 100, SetENOAutomatically false, UDAEnableTagReadback false
   VAR
      Axe_X1 : Struct
         _ActPos : Real;
         _ActVel : Real;
         _Mode : Int;
         Home : Bool;
         Halt : Bool;
         Jog : Bool;
         MoveAbs : Bool;
         MoveRel : Bool;
         MoveVel : Bool;
         PowerOff : Bool;
         PowerOn : Bool;
         SensPos : Bool;
         SensNeg : Bool;
         xBusy : Bool;
         xHomed : Bool;
         xMoveAbsDone : Bool;
         xMoveRelDone : Bool;
         xPower : Bool;
      END_STRUCT;
      Axe_X2 : Struct
         _ActPos : Real;
         _ActVel : Real;
         _Mode : Int;
         Home : Bool;
         Halt : Bool;
         Jog : Bool;
         MoveAbs : Bool;
         MoveRel : Bool;
         MoveVel : Bool;
         PowerOff : Bool;
         PowerOn : Bool;
         SensPos : Bool;
         SensNeg : Bool;
         xBusy : Bool;
         xHomed : Bool;
         xMoveAbsDone : Bool;
         xMoveRelDone : Bool;
         xPower : Bool;
      END_STRUCT;
      Axe_Y : Struct
         _ActPos : Real;
         _ActVel : Real;
         _Mode : Int;
         Home : Bool;
         Halt : Bool;
         Jog : Bool;
         MoveAbs : Bool;
         MoveRel : Bool;
         MoveVel : Bool;
         PowerOff : Bool;
         PowerOn : Bool;
         SensPos : Bool;
         SensNeg : Bool;
         xBusy : Bool;
         xHomed : Bool;
         xMoveAbsDone : Bool;
         xMoveRelDone : Bool;
         xPower : Bool;
      END_STRUCT;
      Axe_Z : Struct
         _ActPos : Real;
         _ActVel : Real;
         _Mode : Int;
         Home : Bool;
         Halt : Bool;
         Jog : Bool;
         MoveAbs : Bool;
         MoveRel : Bool;
         MoveVel : Bool;
         PowerOff : Bool;
         PowerOn : Bool;
         SensPos : Bool;
         SensNeg : Bool;
         xBusy : Bool;
         xHomed : Bool;
         xMoveAbsDone : Bool;
         xMoveRelDone : Bool;
         xPower : Bool;
      END_STRUCT;
   END_VAR
BEGIN

REGION Network 1: Station 3 - Axe X1 (Brushless)
   // //___ ModePose : 
   //          1 ---> Relative positioning
   //          2 ---> Absolute positioning
   //          3 ---> Not supported
   //          4 ---> Referencing - referencing point approach
   //          5 ---> Referencing - set referencing point
   //          6 ---> Traversing block (record mode)
   //          7 ---> Jog
   //          8 ---> Not supported
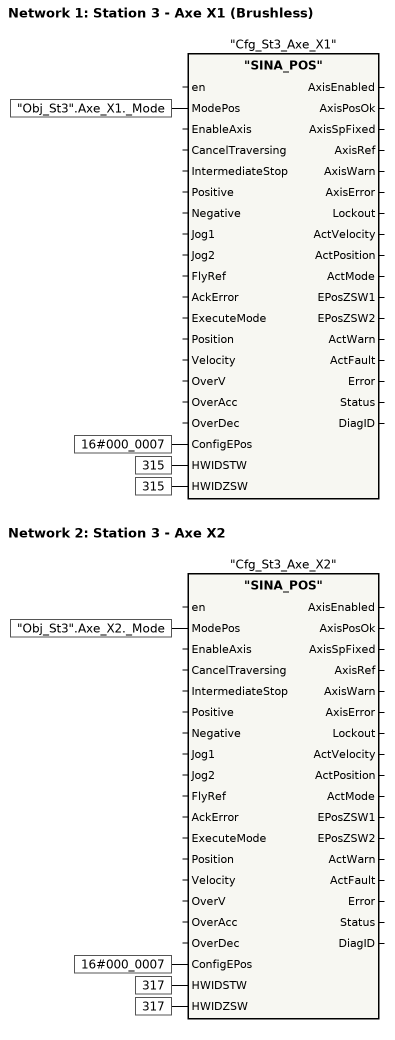
   "Cfg_St3_Axe_X1"(ModePos := "Obj_St3".Axe_X1._Mode,   // "SINA_POS"
                    ConfigEPos := 16#000_0007,
                    HWIDSTW := 315,
                    HWIDZSW := 315);
END_REGION

REGION Network 2: Station 3 - Axe X2
   // //___ ModePose : 
   //          1 ---> Relative positioning
   //          2 ---> Absolute positioning
   //          3 ---> Not supported
   //          4 ---> Referencing - referencing point approach
   //          5 ---> Referencing - set referencing point
   //          6 ---> Traversing block (record mode)
   //          7 ---> Jog
   //          8 ---> Not supported
   "Cfg_St3_Axe_X2"(ModePos := "Obj_St3".Axe_X2._Mode,   // "SINA_POS"
                    ConfigEPos := 16#000_0007,
                    HWIDSTW := 317,
                    HWIDZSW := 317);
END_REGION

REGION Network 3: Station 3 - Axe Y
   // //___ ModePose : 
   //          1 ---> Relative positioning
   //          2 ---> Absolute positioning
   //          3 ---> Not supported
   //          4 ---> Referencing - referencing point approach
   //          5 ---> Referencing - set referencing point
   //          6 ---> Traversing block (record mode)
   //          7 ---> Jog
   //          8 ---> Not supported
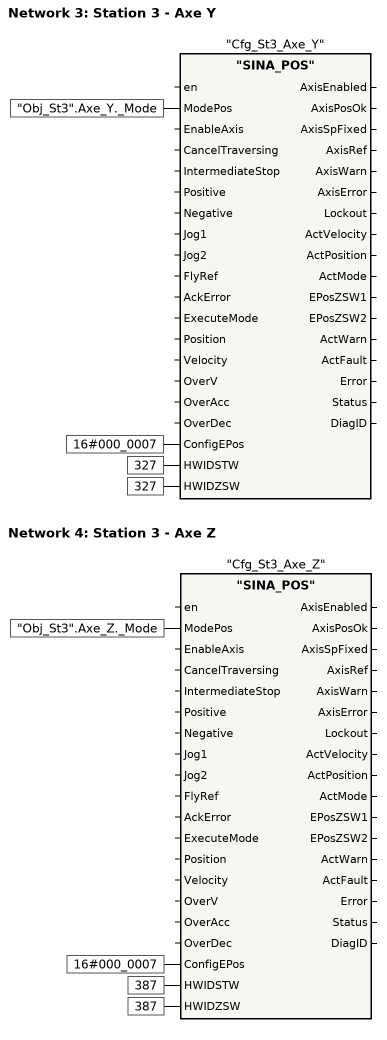
   "Cfg_St3_Axe_Y"(ModePos := "Obj_St3".Axe_Y._Mode, ConfigEPos := 16#000_0007, HWIDSTW := 327, HWIDZSW := 327);   // "SINA_POS"
END_REGION

REGION Network 4: Station 3 - Axe Z
   // //___ ModePose : 
   //          1 ---> Relative positioning
   //          2 ---> Absolute positioning
   //          3 ---> Not supported
   //          4 ---> Referencing - referencing point approach
   //          5 ---> Referencing - set referencing point
   //          6 ---> Traversing block (record mode)
   //          7 ---> Jog
   //          8 ---> Not supported
   "Cfg_St3_Axe_Z"(ModePos := "Obj_St3".Axe_Z._Mode, ConfigEPos := 16#000_0007, HWIDSTW := 387, HWIDZSW := 387);   // "SINA_POS"
END_REGION
END_FUNCTION_BLOCK

FUNCTION_BLOCK "Obj_St4_FB"   // FB400, FBD
{ S7_Optimized_Access := 'TRUE' }
VERSION : 0.1
// stored: AutoNumber false, IsIECCheckEnabled false, IsRetainMemResEnabled false, MemoryReserve 100, SetENOAutomatically false, UDAEnableTagReadback false
   VAR
      Axe_X1 : Struct
         _ActPos : Real;
         _ActVel : Real;
         _Mode : Int;
         Home : Bool;
         Halt : Bool;
         Jog : Bool;
         MoveAbs : Bool;
         MoveRel : Bool;
         MoveVel : Bool;
         PowerOff : Bool;
         PowerOn : Bool;
         SensPos : Bool;
         SensNeg : Bool;
         xBusy : Bool;
         xHomed : Bool;
         xMoveAbsDone : Bool;
         xMoveRelDone : Bool;
         xPower : Bool;
      END_STRUCT;
      Axe_Y1 : Struct
         _ActPos : Real;
         _ActVel : Real;
         _Mode : Int;
         Home : Bool;
         Halt : Bool;
         Jog : Bool;
         MoveAbs : Bool;
         MoveRel : Bool;
         MoveVel : Bool;
         PowerOff : Bool;
         PowerOn : Bool;
         SensPos : Bool;
         SensNeg : Bool;
         xBusy : Bool;
         xHomed : Bool;
         xMoveAbsDone : Bool;
         xMoveRelDone : Bool;
         xPower : Bool;
      END_STRUCT;
      Axe_Y2 : Struct
         _ActPos : Real;
         _ActVel : Real;
         _Mode : Int;
         Home : Bool;
         Halt : Bool;
         Jog : Bool;
         MoveAbs : Bool;
         MoveRel : Bool;
         MoveVel : Bool;
         PowerOff : Bool;
         PowerOn : Bool;
         SensPos : Bool;
         SensNeg : Bool;
         xBusy : Bool;
         xHomed : Bool;
         xMoveAbsDone : Bool;
         xMoveRelDone : Bool;
         xPower : Bool;
      END_STRUCT;
      Prehenseur_Z2 : Struct
         _ActPos : Real;
         _ActVel : Real;
         _Mode : Int;
         Home : Bool;
         Halt : Bool;
         Jog : Bool;
         MoveAbs : Bool;
         MoveRel : Bool;
         MoveVel : Bool;
         PowerOff : Bool;
         PowerOn : Bool;
         SensPos : Bool;
         SensNeg : Bool;
         xBusy : Bool;
         xHomed : Bool;
         xMoveAbsDone : Bool;
         xMoveRelDone : Bool;
         xPower : Bool;
      END_STRUCT;
      Prehenseur_Z3 : Struct
         _ActPos : Real;
         _ActVel : Real;
         _Mode : Int;
         Home : Bool;
         Halt : Bool;
         Jog : Bool;
         MoveAbs : Bool;
         MoveRel : Bool;
         MoveVel : Bool;
         PowerOff : Bool;
         PowerOn : Bool;
         SensPos : Bool;
         SensNeg : Bool;
         xBusy : Bool;
         xHomed : Bool;
         xMoveAbsDone : Bool;
         xMoveRelDone : Bool;
         xPower : Bool;
      END_STRUCT;
   END_VAR
BEGIN

REGION Network 1: Station 4 (Marquage) - Axe X
   // //___ ModePose : 
   //          1 ---> Relative positioning
   //          2 ---> Absolute positioning
   //          3 ---> Not supported
   //          4 ---> Referencing - referencing point approach
   //          5 ---> Referencing - set referencing point
   //          6 ---> Traversing block (record mode)
   //          7 ---> Jog
   //          8 ---> Not supported
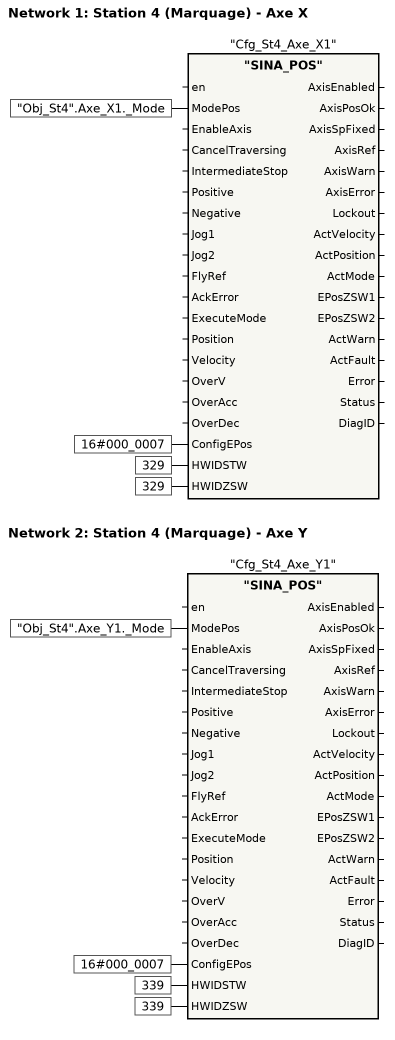
   "Cfg_St4_Axe_X1"(ModePos := "Obj_St4".Axe_X1._Mode,   // "SINA_POS"
                    ConfigEPos := 16#000_0007,
                    HWIDSTW := 329,
                    HWIDZSW := 329);
END_REGION

REGION Network 2: Station 4 (Marquage) - Axe Y
   // //___ ModePose : 
   //          1 ---> Relative positioning
   //          2 ---> Absolute positioning
   //          3 ---> Not supported
   //          4 ---> Referencing - referencing point approach
   //          5 ---> Referencing - set referencing point
   //          6 ---> Traversing block (record mode)
   //          7 ---> Jog
   //          8 ---> Not supported
   "Cfg_St4_Axe_Y1"(ModePos := "Obj_St4".Axe_Y1._Mode,   // "SINA_POS"
                    ConfigEPos := 16#000_0007,
                    HWIDSTW := 339,
                    HWIDZSW := 339);
END_REGION

REGION Network 3: Station 4 (Conforme) - Axe Y
   // //___ ModePose : 
   //          1 ---> Relative positioning
   //          2 ---> Absolute positioning
   //          3 ---> Not supported
   //          4 ---> Referencing - referencing point approach
   //          5 ---> Referencing - set referencing point
   //          6 ---> Traversing block (record mode)
   //          7 ---> Jog
   //          8 ---> Not supported
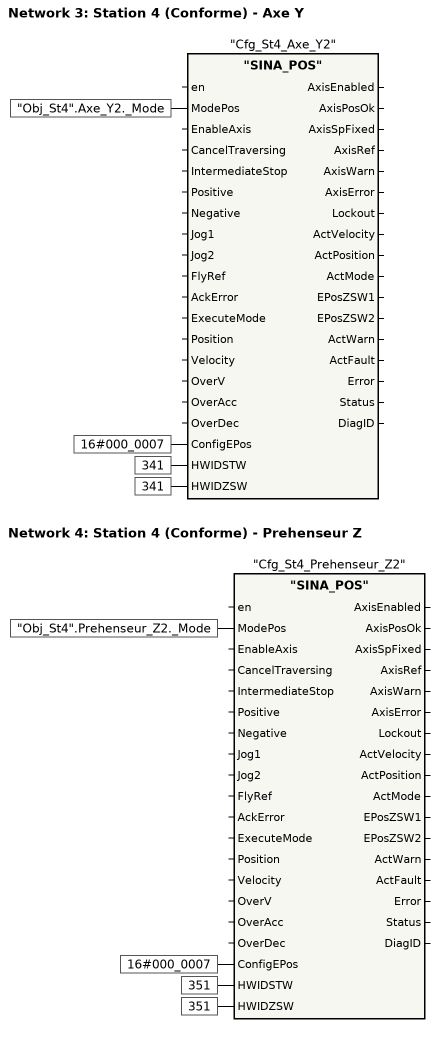
   "Cfg_St4_Axe_Y2"(ModePos := "Obj_St4".Axe_Y2._Mode,   // "SINA_POS"
                    ConfigEPos := 16#000_0007,
                    HWIDSTW := 341,
                    HWIDZSW := 341);
END_REGION

REGION Network 4: Station 4 (Conforme) - Prehenseur Z
   // //___ ModePose : 
   //          1 ---> Relative positioning
   //          2 ---> Absolute positioning
   //          3 ---> Not supported
   //          4 ---> Referencing - referencing point approach
   //          5 ---> Referencing - set referencing point
   //          6 ---> Traversing block (record mode)
   //          7 ---> Jog
   //          8 ---> Not supported
   "Cfg_St4_Prehenseur_Z2"(ModePos := "Obj_St4".Prehenseur_Z2._Mode,   // "SINA_POS"
                           ConfigEPos := 16#000_0007,
                           HWIDSTW := 351,
                           HWIDZSW := 351);
END_REGION

REGION Network 5: Station 4 (Non-Conforme) - Prehenseur Z
   // //___ ModePose : 
   //          1 ---> Relative positioning
   //          2 ---> Absolute positioning
   //          3 ---> Not supported
   //          4 ---> Referencing - referencing point approach
   //          5 ---> Referencing - set referencing point
   //          6 ---> Traversing block (record mode)
   //          7 ---> Jog
   //          8 ---> Not supported
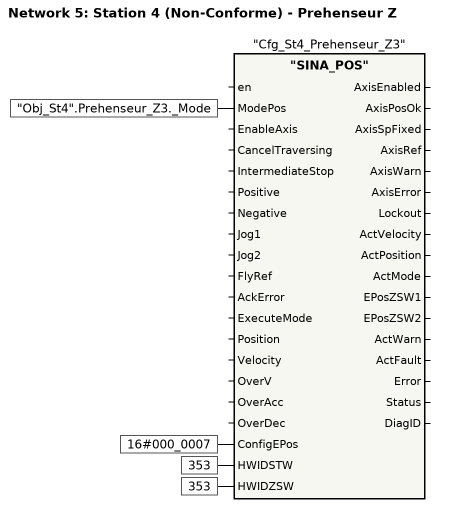
   "Cfg_St4_Prehenseur_Z3"(ModePos := "Obj_St4".Prehenseur_Z3._Mode,   // "SINA_POS"
                           ConfigEPos := 16#000_0007,
                           HWIDSTW := 353,
                           HWIDZSW := 353);
END_REGION
END_FUNCTION_BLOCK

FUNCTION_BLOCK "SINA_INFEED"
TITLE = 'operate a line module'
{ S7_Optimized_Access := 'TRUE' }
AUTHOR : DRVDPS7
FAMILY : DRIVES
NAME : SINA_INFEED
VERSION : 5.2
//Control basic infeed
   VAR_INPUT 
      EnablePrecharging : Bool;   // 0-->1 = Setup the DC Link (BLM/SLM/ALM) (OFF1 = 0-->1)
      EnableInfeed : Bool;   // 1 = Enable "active" line modules  (only SLM / ALM)
      AckFault : Bool;   // 1 = Acknowledge infeed error
      ConfigAxis : Word := 16#0001;   // binary programmed input to control all functions in the telegram without its own function block input
      HWIDSTW : HW_IO;   // Hardware Identifer set point slot
      HWIDZSW : HW_IO;   // Hardware Identifer actual value slot
   END_VAR

   VAR_OUTPUT 
      Ready { ExternalVisible := 'False'} : Bool;   // 1 = Infeed ready to power up
      Operation { ExternalVisible := 'False'} : Bool;   // 1 = Infeed ready for operation
      Run { ExternalVisible := 'False'} : Bool;   // 1 = Infeed in operation (only SLM / ALM)
      Fault { ExternalVisible := 'False'} : Bool;   // 1 = Infeed error active
      Lockout { ExternalVisible := 'False'} : Bool;   // 1 = Infeed lockout active
      Warning { ExternalVisible := 'False'} : Bool;   // 1 = Infeed warning active
      ZSW1 : Word := 16#0000;   // Infeed Status word
      Error { ExternalVisible := 'False'} : Bool;   // Rising edge informs that an error occurred during the execution of
      Status : Word := #STATUS_SUBSEQUENT_CALL;   // Status output (7002 = FB in operation; 8xxx = error description  - read the manual)
      DiagID : Word;   // Error codes of the cyclic system funtion blocks DPWR / DPRD_DAT
   END_VAR

   VAR 
      statStwOnOff : Bool;   // STW 1.0
      statStwOff2 : Bool;   // STW 1.1
      statStwQuickStop : Bool;   // STW 1.2
      statStwOperation : Bool;   // STW 1.3
      statStwReleaseRunup : Bool;   // STW 1.4
      statStwDisMotOp : Bool;   // STW 1.5
      statStwDisRegOp : Bool;   // STW 1.6
      statStwAckFault : Bool;   // STW 1.7
      statStwConductRequested : Bool;   // STW 1.10
      statStwDirectOfRot : Bool;   // STW 1.11
      statSTW1 : Word := 16#0062;
      statReady : Bool;
      statOperation : Bool;
      statRun : Bool;
      statFault : Bool;
      statLockout : Bool;
      statWarning : Bool;
   END_VAR

   VAR_TEMP 
      tempRetValDPRD : Int;   // Temporary value for infeed enabled
      tempRetValDPWR : Int;
   END_VAR

   VAR CONSTANT 
      STATUS_SUBSEQUENT_CALL : Word := 16#7002;   // Subsequent call of FB
      STATUS_WARN_INFEED : Word := 16#7200;   // Infeed warning active
      STATUS_ERROR_PRE : Word := 16#8400;   // Infeed error with the precharge step
      STATUS_ERROR_INF : Word := 16#8401;   // Infeed error (general)
      STATUS_ERROR_DPRD_DAT : Word := 16#8600;   // Error "Read cyclic data" operation
      STATUS_ERROR_DPWR_DAT : Word := 16#8601;   // Error "Write cyclic data" operation
   END_VAR


BEGIN
	//=============================================================================
	//SIEMENS AG
	//(c)Copyright 2017 All Rights Reserved
	//-----------------------------------------------------------------------------
	// Library: DriveLib
	// Tested with: S7-1516-3 PN/DP V1.8
	// Engineering: TIA Portal V14
	// Restrictions: -
	// Requirements: S7-1200 / S7-1500
	// Functionality: the block serves to supply a rectifier unit line module
	//-----------------------------------------------------------------------------
	// Change log table:
	// Version Date       Expert in charge Changes applied
	// 0.1     28.09.2015 ZP               First released version
	// 0.2     09.11.2015 ZP               no internal acknowledgment
	// 0.3     30.11.2015 ZP               new input parameter ConfigAxis
	// 5.0     11.01.2017 FG               adapt version to new DriveLib version
	// 5.1     02.05.2018 FG               Connect all bits from ConfigAxis with
	//                                     the Bits from STW1
	// 5.2     10.06.2021 FG               Error correction RQ 5680664
	//=============================================================================
	
	// presetting STW1
	#statStwOnOff := FALSE;     // STW1.0
	#statStwOperation := FALSE;     // STW1.3
	#statStwAckFault := FALSE;      // STW1.7
	#statStwConductRequested := true; //STW1.10 conduct requested set cyclic
	
	// external setting of STW1
	#statStwOff2 := #ConfigAxis.%X0;  // TRUE if "ConfigAxis" is not assigned STW1.1
	
	#statStwDisMotOp := #ConfigAxis.%X2;  // TRUE if "ConfigAxis" is not assigned STW1.5
	#statStwDisRegOp := #ConfigAxis.%X3; // TRUE if "ConfigAxis" is not assigned STW1.6
	
	// reset error
	#Error := FALSE;
	// acknowledge fault?
	
	IF #AckFault THEN
	  #statStwAckFault := TRUE;  // input AckFault into STW1.7
	END_IF;
	
	// read status word
	#tempRetValDPRD := DPRD_DAT(LADDR := #HWIDZSW, RECORD => #ZSW1);
	
	//==========================================
	//#ZSW1 := "SIM_ZSW1";  // only for test
	//==========================================
	
	// write status word into static word
	#statReady := #ZSW1.%X0;
	#statOperation := #ZSW1.%X1;
	#statRun := #ZSW1.%X2;
	#statFault := #ZSW1.%X3;
	#statLockout := #ZSW1.%X6;
	#statWarning := #ZSW1.%X7;
	
	// write status word to output
	#Ready := #statReady;
	#Operation := #statOperation;
	#Run := #statRun;
	#Fault := #statFault;
	#Lockout := #statLockout;
	#Warning := #statWarning;
	
	// Check preconditions
	IF #EnablePrecharging AND #Ready AND NOT #Lockout AND NOT #Fault THEN
	  #statStwOnOff := TRUE;      // STW1.0 
	  //  #statStwAckFault := FALSE;      // STW1.7
	END_IF;
	
	IF #EnablePrecharging AND #Ready AND NOT #Lockout AND NOT #Fault AND NOT #EnableInfeed THEN
	  #statStwOperation := FALSE;     // STW1.3
	END_IF;
	
	IF #EnablePrecharging AND #Ready AND NOT #Lockout AND NOT #Fault AND #EnableInfeed AND NOT #Operation THEN
	  #statStwOperation := FALSE;     // STW1.3
	END_IF;
	
	IF #EnablePrecharging AND #Ready AND NOT #Lockout AND NOT #Fault AND #EnableInfeed AND #Ready AND #Operation THEN
	  #statStwOperation := TRUE;     // STW1.3
	END_IF;
	
	//Error handling and diagnistic DPRD_DAT / DPWR_DAT 
	#Status := #STATUS_SUBSEQUENT_CALL;     // no error activ 16#7002
	
	IF (NOT #EnablePrecharging AND #EnableInfeed) THEN
	  #Error := TRUE;
	  #Status := #STATUS_ERROR_PRE; // error precharching 16#8400
	  #statStwOperation := FALSE;     // STW1.3 
	  #statStwOnOff := FALSE;     // STW1.0
	END_IF;
	
	IF (NOT #EnablePrecharging AND NOT #EnableInfeed) THEN
	  #statStwOperation := FALSE;     // STW1.3 
	  #statStwOnOff := FALSE;     // STW1.0
	END_IF;
	
	// write control word - internal 
	#statSTW1.%X0 := #statStwOnOff;
	#statSTW1.%X3 := #statStwOperation;
	#statSTW1.%X7 := #statStwAckFault;
	#statSTW1.%X10 := #statStwConductRequested;
	// write control word - external 
	#statSTW1.%X1 := #statStwOff2;
	#statSTW1.%X2 := #ConfigAxis.%X4;
	#statSTW1.%X4 := #ConfigAxis.%X5;
	#statSTW1.%X5 := #statStwDisMotOp;
	#statSTW1.%X6 := #statStwDisRegOp;
	#statSTW1.%X8 := #ConfigAxis.%X6;
	#statSTW1.%X9 := #ConfigAxis.%X7;
	#statSTW1.%X11 := #ConfigAxis.%X8;
	#statSTW1.%X12 := #ConfigAxis.%X9;
	#statSTW1.%X13 := #ConfigAxis.%X10;
	#statSTW1.%X14 := #ConfigAxis.%X11;
	#statSTW1.%X15 := #ConfigAxis.%X12;
	
	#tempRetValDPWR := DPWR_DAT(LADDR := #HWIDSTW, RECORD := #statSTW1); // write STW1
	
	#DiagID := 16#0;
	
	IF #Warning THEN
	  #Status := #STATUS_WARN_INFEED;     // warning infeed 16#7200
	ELSIF #Fault THEN
	  #Status := #STATUS_ERROR_INF;       // error infeed 16#8401
	ELSIF #tempRetValDPRD <> 16#0 THEN
	  #Status := #STATUS_ERROR_DPRD_DAT;       // error code DPRD_DAT 16#8600
	  #DiagID := INT_TO_WORD(#tempRetValDPRD);        // diagnistic DPRD_DAT
	  #Error := TRUE;
	ELSIF #tempRetValDPWR <> 16#0 THEN
	  #Status := #STATUS_ERROR_DPWR_DAT;       // error code DPWR_DAT 16#8601
	  #DiagID := INT_TO_WORD(#tempRetValDPWR);        // diagnistic DPWR_DAT
	  #Error := TRUE;
	END_IF;
	
	
	
	
	
END_FUNCTION_BLOCK

FUNCTION_BLOCK "SINA_PARA"
TITLE = 'parameter exchange between SINAMICS and S7'
{ S7_Optimized_Access := 'TRUE' }
AUTHOR : DRVDPS7
FAMILY : DRIVES
NAME : SINA_PAR
VERSION : 5.1
//Copyright (C) Siemens AG 2012. All Rights Reserved. Confidential
//--------------------------------------------------------------------------- 
//SINA_PARA: Austausch 15 beliebiger Parameter zwischen SINAMICS S120/G120 <-> S7
//-------------------------------------------------------------------------- Ersteller: Siemens AG Erlangen A&D MC PM   Datum:  07.07.10        Vers.:2.1
//Änderung:  J.B. Typical Team                       09.01.13              2.2
//    Umsetzung in SCL / TIA 
//Änderung:  J.B. Typical Team                       29.04.13              2.3 
//    "Q" an den Ausgänge entfernen
//     
//Änderung:  J.B. Typical Team                       28.06.13              2.4
//    HW-Zugriffsermittlung über LOG2MOD
//
//Änderung:  J.B. Typical Team                       25.07.13              2.5
//    Wiederholfaktor bei temporäre Fehler
//        
//Änderung:  J.B. Typical Team                       24.09.13              2.6
//    Konvertierungsfehler
//    
//Änderung:  J.B. Typical Team                       05.10.13              2.7
//    Fehlerkorrektur im Antworttelegramm bei 
//    Änderung
//Änderung:  J.B. Typical Team                       16.12.13              2.8
//    weiterhin Fehlerkorrektur im Antworttelegramm bei 
//    Änderung
//    
//Änderung:  J.B. Typical Team                       15.01.14              2.9
//    weiterhin Fehlerkorrektur im Antworttelegramm bei 
//    Änderung
//Änderung:  J.B. Typical Team                       17.07.14              3.0
//    Nun mit Optimierung 
//
//Änderung:  J.B. Typical Team                       30.07.14              4.0
//    Festlegung auf einheitlicher neuer Version 4.0
//
//Änderung:  G.F. Typical Team                       20.05.15              4.1
//    Fehler bei der Umrechnung der Parameterwerte behoben
//
//Änderung:  G.F. Typical Team                       15.09.15              4.2
//    Defaultwert des Parameters AxisNo von 0 auf 1 geändert
//
//Änderung:  G.F. Typical Team                       06.10.15              4.3
//    Defaultwert der Parameter AxisNo, ParaNo und Done von 0 auf 1 geändert
//    und Parameter swParaError gezielt auf 0 gesetzt
//
//Änderung:  J.B. Typical Team                       08.12.15              4.4
//    1. Wenn beim Parameter "Lesen" ein Fehler zurück gemeldet wird, 
//    soll das "Schreiben" abgebrochen werden
//
//    2. Für den Datentyp DWORD mit/ohne Vorzeichen neuer Ablageort
//    (statt REAL nun DINT)
//
//    3. Neue Ausgangsvariable Ready = Lesen/Schreiben der Parameter
//    abgeschlossen
//
//    4. Austauch der Parameter kann jetzt abgebrochen werden
//
//    5. Warnung durch Initialisierung elimininiert
//
//    6. Eingang Laddr in hardwareId umbenannt
//
//Änderung:  G.F. Typical Team                       24.11.16              4.5
//    - Fehlerausgabe bei unbekannten Datentyp (ErrorId := 5)
//    - Datentyp 10 (OctetString) wird unterstützt
//    - Datentyp 13 (TimeDifference) wird unterstützt
//    - Fehler bei Auftrag abbrechen behoben
//
//Änderung:  G.F. Typical Team                       11.01.17              5.0
//    - Festlegung auf einheitlicher neuer Version 5.0 
//
//Bibliothek V7
//Funktion: Austausch 15 beliebiger Parameter zwischen SINAMICS S120/G120 <-> S7
//********************************************************************************************************************************************************
//************************************************************************FB283***************************************************************************
//********************************************************************************************************************************************************
   VAR_INPUT 
      Start { CFC_Visible := 'true'; CFC_ForTest := 'true'} : Bool := 0;   // Start of the job (0 = no job or cancel the actual job; 1= start job and perform the job)
      ReadWrite { CFC_Visible := 'true'; CFC_ForTest := 'true'} : Bool := 0;   // Type of job 0 = read parameter, 1 = write parameter
      ParaNo { CFC_Visible := 'true'; CFC_ForTest := 'true'} : Int := 1;   // Number of parameters to read or write
      AxisNo { CFC_Visible := 'true'; CFC_ForTest := 'true'} : Byte := 16#01;   // Object ID of drive Output variables
      hardwareId : HW_IO := 0;   // Configured diagnosis address of the module (DEC) for WRREC and RDREC
   END_VAR

   VAR_OUTPUT 
      Ready { CFC_Visible := 'true'; CFC_ForTest := 'true'} : Bool := 0;   // Read or write parameter order ready
      Busy { CFC_Visible := 'true'; CFC_ForTest := 'true'} : Bool := 0;   // =1 Mode of operation is explained
      Done { CFC_Visible := 'true'; CFC_ForTest := 'true'} : Bool := 1;   // =1 Mode of operation without mistake finishes
      Error { CFC_Visible := 'true'; CFC_ForTest := 'true'} : Bool := 0;   // Error or faults are active
      ErrorId { CFC_Visible := 'true'; CFC_ForTest := 'true'} : DWord := 0;   // Mode of operation disturbance
      DiagId { CFC_Visible := 'true'; CFC_ForTest := 'true'} : Word := 16#0000;   // Extended communication errorStatic variables
   END_VAR

   VAR 
      sbWrError : Bool := 0;   // Error when writing with SFB WRREC
      sbWrDone : Bool := 0;   // Data record written with SFB WRREC
      sbRdError : Bool := 0;   // Error when reading with SFB RDREC
      sbWrBusy : Bool := 0;   // Write Task busy SFB 53 WRREC
      sbRdBusy : Bool := 0;   // Read Task busy SFB 52 RDREC
      sbWrStart : Bool := 0;   // Start write job
      sbRdStart : Bool := 0;   // Start read job
      sbWrStart1 : Bool := 0;   // Start write job (first part of write commando)
      sbRdStart1 : Bool := 0;   // Start read job (first part of read commando)
      sbWrStart2 : Bool := 0;   // Start write job (second part of write commando)
      sbRdStart2 : Bool := 0;   // Start read job (second part of read commando)
      sbStart : Bool := 0;   // Positive edge of Start commando
      sbReady : Bool := 0;   // Positive edge of Ready
      sbRead : Bool := 0;   // Commando "Read"
      sbWrite : Bool := 0;   // Commando "Write"
      sbParaNo : Bool := 0;   // The count of parameter are Okay
      sbBusy : Bool := 0;   // Mode of operation is explained
      sbError : Bool := 0;   // Error or faults are active
      sbDone : Bool := 0;   // Job finished
      siParaNo : Int := 0;   // Count of parameter are read or write
      syAxisNo : Byte := 0;   // Axis ID
      siReqRef : Int := 0;   // Reference number of request
      siErrorId : Int := 0;   // Function block fault ID
      siErrorCount : Int := 0;   // temporary error counter of retry job
      siMaxErrCount : Int := 12500;   // max. temporary error counter
      swParaError : Word := WORD#16#0000;   // Error of parameter
      sxReqParaMulti : Struct   // Telegramm for request/change parameter value, multi-parameter
         sxHeader : Struct   // Request header
            syReqRef : Byte := 16#00;   // Request reference (Request ID, mirrored in response)
            syReqId : Byte := 16#01;   // Request ID 0x1=Read
            syAxisNo : Byte := 16#00;   // Axis (0x0=Axis A | 0x1=Axis B)
            syParaNo : Byte := 16#00;   // No. of parameters (DEC: for single parameters=1)
         END_STRUCT;
         sxParaAdress : Array[1..16] of Struct   // Parameter address 1..16
            syAttr : Byte := 16#10;   // Attribute of parameters (0x10=Value, 0x30=Text)
            syElemNo : Byte := 16#01;   // No. of elements (DEC: for single elements=1)
            siParaNo : UInt := 0;   // Number of parameter (Number 1..65535)
            siIndex : UInt := 0;   // Subindex (Number 1..65535)
         END_STRUCT;
      END_STRUCT;
      sxChaParaMulti : Struct   // Telegramm for change parameter value, multi-parameter
         sxHeader : Struct   // Request header
            syReqRef : Byte := 16#00;   // Request reference (Request ID, mirrored in response)
            syReqId : Byte := 16#02;   // Request ID 0x2=Write
            syAxisNo : Byte := 16#00;   // Axis (0x0=Axis A | 0x1=Axis B)
            syParaNo : Byte := 16#00;   // No. of parameters (DEC: for single parameters=1)
         END_STRUCT;
         sxData : Array[1..192] of Byte;   // Parameter address 1..16 (Attribute/Value (BYTE), Number of Elements (BYTE), Parameter number (2 BYTES), Subindex (2 BYTES), Parameter value 1..16 (Format/Error (BYTE), Number of Values/Value of Error (BYTE), Value (BYTE or WORD or DWORD)
      END_STRUCT;
      sxRespParaMulti : Struct   // Telegramm for response parameter value, multi-parameter
         sxHeader : Struct   // Request header
            syReqRef : Byte := 16#00;   // Request reference (Request ID, mirrored in response)
            syReqId : Byte := 16#00;   // Request ID (0x1=Read | 0x2=Write)
            syAxisNo : Byte := 16#00;   // Axis (0x0=Axis A | 0x1=Axis B)
            syParaNo : Byte := 16#00;   // No. of parameters (DEC: for single parameters=1)
         END_STRUCT;
         sxData : Array[1..96] of Byte;   // Parameter value 1..16 (Format/Error (BYTE), Number of Values/Value of Error (BYTE), Value (BYTE or WORD or DWORD)
      END_STRUCT;
      sxParameter : Array[1..16] of Struct   // List of parameter (max. 16 parameter)
         siParaNo : UInt := 0;   // Number of parameter (Number 1..65535)
         siIndex : UInt := 0;   // Subindex (Number 1..65535)
         srValue : Real := 0.0;   // Value of parameter
         sdValue : DInt := 0;   // Value of parameter
         syFormat : Byte := BYTE#16#00;   // Format of value (Format 0x40..0x44)
         swErrorNo : Word := WORD#16#0000;   // Error number (see table below)
      END_STRUCT;
      RDREC_1 {InstructionName := 'RDREC'; LibVersion := '1.0'} : RDREC;
      WRREC_1 {InstructionName := 'WRREC'; LibVersion := '1.1'} : WRREC;
      siParaNoMax : Int := 16;   // max. Anzahl der Parameter
      siLenHeader : Int := 4;   // Length of telegram of header
      siLenParaMulti : Int := 96;   // Length of telegram of data for request and response
      siLenChaPara : Int := 192;   // Length of telegram of data for change parameterTemporary variables
   END_VAR

   VAR_TEMP 
      piCount : Int;   // Freely available counter variable
      piPointer : Int;   // Freely available pointer array variable
      piLenTele : Int;   // Length of telegram of buffer
      piRetSFC : Int;   // Status for fault analysis
      pwWordHigh : Word;   // Help variable of word
      pwWordLow : Word;   // Help variable of word
      pwWord1 : Word;   // Help variable of word
      pwWord2 : Word;   // Help variable of word
      pdDWordHigh : DWord;   // Help variable of dword
      pdDWordLow : DWord;   // Help variable of dword
      pdStatus : DWord;   // Status[1] = Error => Status[2] Error Decode + Status[3] Error Code
      pbValidSFB : Bool;   // Status SFB
      piLenSFB : UInt;   // Status length for SFB call
      pwErrorNo : Word;   // Error number
   END_VAR


BEGIN
	
	//=============================================================================
	//SIEMENS AG
	//(c)Copyright 2017 All Rights Reserved
	//-----------------------------------------------------------------------------
	// Library: DriveLib
	// Tested with: S7-1516-3 PN/DP V1.8
	// Engineering: TIA Portal V14
	// Restrictions: -
	// Requirements: S7-1200 / S7-1500
	// Functionality: read and write up to 15 parameter from/to a Sinamics
	//
	//=============================================================================
	
	// Auftrag "Parameter lesen" bzw. Auftrag "Parameter schreiben" wird nicht mehr ausgeführt
	IF NOT #sbBusy THEN
	  // Überprüfung der auf korrekte Parametrierung der Anzahl der Parameter
	  IF #ParaNo > #siParaNoMax THEN
	    
	    #sbParaNo := FALSE;
	    #sbError := True;
	    #siErrorId := 2;
	  ELSIF #ParaNo < 1 THEN
	    
	    #sbParaNo := FALSE;
	    #sbError := True;
	    #siErrorId := 2;
	  ELSE
	    
	    #sbParaNo := TRUE;
	    #siParaNo := #ParaNo;
	    
	    IF #siErrorId = 2 THEN
	      #siErrorId := 0;
	      #sbError := False;
	    END_IF;
	  END_IF;
	  
	  #syAxisNo := #AxisNo;
	END_IF;
	
	// Starten 
	IF #Start AND NOT #sbStart AND (#ParaNo <> 0) AND NOT #sbBusy THEN
	  
	  #sbReady := False;
	  #sbError := False;
	  #sbBusy := False;
	  
	  // Auftrag "Parameter lesen" erkennen
	  IF NOT #ReadWrite THEN
	    #sbRead := True;
	    #sbWrStart := True;
	    #sbRdStart := False;
	    
	    #sbWrite := False;
	    #sbWrStart1 := False;
	    #sbRdStart1 := False;
	    #sbWrStart2 := False;
	    #sbRdStart2 := False;
	    
	    // Referenzauftragsnummer erzeugen
	    #siReqRef := #siReqRef + 1;
	    
	    // bei Überschreitung wieder zurücksetzen und von vorne (Wertebereich von 0-255)
	    IF #siReqRef > 255 THEN
	      #siReqRef := 0;
	    END_IF;
	    
	    // Auftrag "Parameter schreiben" erkennen
	  ELSE
	    #sbWrite := True;
	    #sbWrStart1 := True;
	    #sbRdStart1 := False;
	    #sbWrStart2 := False;
	    #sbRdStart2 := False;
	    
	    #sbRead := False;
	    #sbWrStart := False;
	    #sbRdStart := False;
	    
	    // Referenzauftragsnummer erzeugen
	    #siReqRef := #siReqRef + 1;
	    
	    // bei Überschreitung wieder zurücksetzen und von vorne (Wertebereich von 0-255)
	    IF #siReqRef > 255 THEN
	      #siReqRef := 0;
	    END_IF;
	  END_IF;
	  
	  // Fehler 4 und 5 wieder zurücknehmen
	  IF (#siErrorId = 4) OR (#siErrorId = 5) THEN
	    #sbError := False;
	    #siErrorId := 0;
	  END_IF;
	END_IF;
	
	// "Start commando" Flanke merken
	#sbStart := #Start;
	
	// Abbrechen
	IF NOT #Start THEN
	  
	  #siErrorCount := 0;
	  // Schreib - oder Lesevorgang abbrechen
	  #sbRead := False;
	  #sbWrStart := False;
	  #sbRdStart := False;
	  
	  #sbWrite := False;
	  #sbWrStart1 := False;
	  #sbRdStart1 := False;
	  #sbWrStart2 := False;
	  #sbRdStart2 := False;
	  
	  // Auftag ist noch beschäftigt => Fehler ausgeben
	  IF #sbBusy THEN
	    #sbError := True;
	    #siErrorId := 4;
	    #sbBusy := False;
	  END_IF;
	END_IF;
	
	// Auftrag "Parameter lesen" wurde ausgelöst
	IF #sbParaNo AND #sbRead AND NOT #sbWrite THEN
	  
	  // Auftrag "Parameter lesen" vorbereiten und abschicken
	  IF #sbWrStart THEN
	    
	    // Ablöschen des Sendepuffers
	    IF NOT (#siParaNo = #siParaNoMax) THEN
	      FOR #piCount := #siParaNo TO #siParaNoMax DO
	        
	        // Parameternummer des Parameters 
	        #sxReqParaMulti.sxParaAdress[#piCount].siParaNo := 0;
	        
	        // Subindex des Parameters
	        #sxReqParaMulti.sxParaAdress[#piCount].siIndex := 0;
	      END_FOR;
	    END_IF;
	    
	    // Auftrags-HEADER erstellen
	    // Auftragsreferenz
	    #sxReqParaMulti.sxHeader.syReqRef := INT_TO_BYTE(#siReqRef);
	    
	    // Auftragskennung 0x01=Request Parameters
	    #sxReqParaMulti.sxHeader.syReqId := B#16#01;
	    
	    // Achse
	    #sxReqParaMulti.sxHeader.syAxisNo := #syAxisNo;
	    
	    // Anzahl Parameter        
	    #sxReqParaMulti.sxHeader.syParaNo := INT_TO_BYTE(#siParaNo);
	    
	    // Auftrags-PARAMETERADRESSE erstellen
	    FOR #piCount := 1 TO #siParaNo DO
	      
	      // Parameternummer des Parameters                                
	      #sxReqParaMulti.sxParaAdress[#piCount].siParaNo := #sxParameter[#piCount].siParaNo;
	      
	      // Subindex des Parameters
	      #sxReqParaMulti.sxParaAdress[#piCount].siIndex := #sxParameter[#piCount].siIndex;
	    END_FOR;
	    
	    // SCHREIBEN AZYKLISCH
	    #piLenTele := #siLenHeader + #siLenParaMulti;
	    #WRREC_1(REQ := True,                                // Startimpuls
	             ID := #hardwareId,                         // Diagnoseadresse
	             INDEX := 47,                                  // Rahmentyp
	             LEN := INT_TO_UINT(#piLenTele),             // maximale Länge
	             DONE => #sbWrDone,                           // Schreibauftrag beendet
	             BUSY => #sbWrBusy,                           // Slave beschäftigt
	             ERROR => #sbWrError,                          // Fehler beim Schreiben
	             STATUS => #pdStatus,                           // Status[1] = Error => Status[2] Error Decode + Status[3] Error Code
	             RECORD := #sxReqParaMulti);                    // Zeiger auf zu schreibenen Datensatzes
	    
	    // Ausgänge setzen
	    #sbBusy := #sbWrBusy;
	    #sbDone := #sbWrDone;
	    
	    // Fehler auswerten
	    IF #sbWrError THEN
	      
	      // Fehlerstatus aus dem Doppelwort filtern und weitergeben                
	      #pwWord1 := DWORD_TO_WORD(SHR(IN := (#pdStatus AND DW#16#FFFF00), N := 8));
	      
	      // Fehlerstatus setzen
	      #siErrorId := 3;
	      #DiagId := #pwWord1;
	      
	      //Temporärer Fehler: #pdStatus = 80A7, 80B5, 80C0, 80C1, 80C2, 80C3 oder 80C4 zulassen und nocheinmal versuchen
	      IF NOT (#pwWord1 = DW#16#80A7) AND NOT (#pwWord1 = DW#16#80B5) AND NOT (#pwWord1 = DW#16#80C0) AND
	        NOT (#pwWord1 = DW#16#80C1) AND NOT (#pwWord1 = DW#16#80C2) AND NOT (#pwWord1 = DW#16#80C3) AND
	        NOT (#pwWord1 = DW#16#80C4) THEN
	        
	        // Wiederholungsauftrag wieder zurücknehmen 
	        #sbWrStart := False;
	        #sbRdStart := False;
	        #sbRead := False;
	        
	        // Fehler ausgeben 
	        #sbError := #sbWrError;
	        
	      ELSE
	        // Fehlerwiederholauftrag ??                   
	        IF #siErrorCount = #siMaxErrCount THEN
	          
	          // Wiederholungsauftrag wieder zurücknehmen
	          #sbWrStart := False;
	          #sbRdStart := False;
	          #sbRead := False;
	          
	          //Fehlerzähler zurücksetzen
	          #siErrorCount := 0;
	          
	          // Fehler ausgeben 
	          #sbError := #sbWrError;
	          
	          // nix tun bis Zähler überläuft
	        ELSE
	          #siErrorCount := #siErrorCount + 1;
	        END_IF;
	      END_IF;
	      
	      // kein Fehler beim SCHEIBEN AZYKLISCH und Auftrag fertig 
	    ELSIF NOT #sbWrBusy AND #sbWrDone THEN
	      
	      // Fehlerkennung zurücknehmen
	      IF #siErrorId = 3 THEN
	        #siErrorId := 0;
	        #sbError := False;
	      END_IF;
	      
	      #DiagId := W#16#00;
	      
	      // Schreibauftrag fertig melden und Leseantrag anstossen
	      #sbWrStart := False;
	      #sbRdStart := True;
	    END_IF;
	  END_IF; // Auftrag "Parameter lesen" vorbereiten und abschicken
	  
	  // vom Auftrag "Parameter lesen" die Antwort abwarten und dann auswerten
	  IF #sbRdStart THEN
	    
	    // Ablöschen des Empfangspuffers
	    #sxRespParaMulti.sxHeader.syReqRef := B#16#00;
	    #sxRespParaMulti.sxHeader.syReqId := B#16#00;
	    #sxRespParaMulti.sxHeader.syAxisNo := B#16#00;
	    #sxRespParaMulti.sxHeader.syParaNo := B#16#00;
	    
	    FOR #piCount := 1 TO #siLenParaMulti DO
	      #sxRespParaMulti.sxData[#piCount] := B#16#00;
	    END_FOR;
	    
	    // LESEN AZYKLISCH
	    #piLenTele := #siLenHeader + #siLenParaMulti;
	    #RDREC_1(REQ := True,                                // Startimpuls
	             ID := #hardwareId,                         // Diagnoseadresse        
	             INDEX := 47,                                  // Rahmentyp           
	             MLEN := INT_TO_UINT(#piLenTele),             // maximale Länge
	             VALID => #pbValidSFB,                         // neuer Datensatz empfangen und gültig   
	             BUSY => #sbRdBusy,                           // Slave beschäftigt
	             ERROR => #sbRdError,                          // Fehler beim Schreiben
	             STATUS => #pdStatus,                           // Status[1] = Error => Status[2] Error Decode + Status[3] Error Code 
	             LEN => #piLenSFB,                           // Länge des gelesenen Datensatzes
	             RECORD := #sxRespParaMulti);                   // Zeiger auf gelesenen Datensatz
	    
	    // Ausgänge setzen
	    #sbBusy := #sbRdBusy;
	    #sbDone := #pbValidSFB;
	    
	    // Fehler auswerten
	    IF #sbRdError THEN
	      // Fehlerstatus aus dem Doppelwort filtern und weitergeben                
	      #pwWord1 := DWORD_TO_WORD(SHR(IN := (#pdStatus AND DW#16#FFFF00), N := 8));
	      
	      // Fehlerstatus setzen
	      #siErrorId := 3;
	      #DiagId := #pwWord1;
	      
	      //Temporärer Fehler: #pdStatus = 80A7, 80B5, 80C0, 80C1, 80C2, 80C3 oder 80C4 zulassen und nocheinmal versuchen
	      IF NOT (#pwWord1 = DW#16#80A7) AND NOT (#pwWord1 = DW#16#80B5) AND NOT (#pwWord1 = DW#16#80C0) AND
	        NOT (#pwWord1 = DW#16#80C1) AND NOT (#pwWord1 = DW#16#80C2) AND NOT (#pwWord1 = DW#16#80C3) AND
	        NOT (#pwWord1 = DW#16#80C4) THEN
	        
	        // Wiederholungsauftrag wieder zurücknehmen  
	        #sbWrStart := False;
	        #sbRdStart := False;
	        #sbRead := False;
	        
	        // Fehler ausgeben 
	        #sbError := #sbRdError;
	        
	      ELSE
	        // Fehlerwiederholauftrag ??                   
	        IF #siErrorCount = #siMaxErrCount THEN
	          
	          // Wiederholungsauftrag wieder zurücknehmen
	          #sbWrStart := False;
	          #sbRdStart := False;
	          #sbRead := False;
	          
	          //Fehlerzähler zurücksetzen
	          #siErrorCount := 0;
	          
	          // Fehler ausgeben 
	          #sbError := #sbRdError;
	          
	          // nix tun bis Zähler überläuft
	        ELSE
	          #siErrorCount := #siErrorCount + 1;
	        END_IF;
	      END_IF;
	      
	      // Fehler : die Auftragsreferenz der Antwort übertimmt nicht mit der Auftragsreferenz der Anfrage überein
	    ELSIF NOT (#siReqRef = BYTE_TO_INT(#sxRespParaMulti.sxHeader.syReqRef)) AND NOT #sbRdBusy AND #pbValidSFB THEN
	      #siErrorId := 1;
	      #sbError := True;
	      #sbDone := False;
	      
	      // Wiederholungsauftrag wieder zurücknehmen  
	      #sbWrStart := False;
	      #sbRdStart := False;
	      #sbRead := False;
	      
	      // Fehler : falsche Auftragskennung zurück erhalten    
	    ELSIF NOT (#sxRespParaMulti.sxHeader.syReqId = B#16#81 OR #sxRespParaMulti.sxHeader.syReqId = B#16#01) AND
	      NOT #sbRdBusy AND #pbValidSFB THEN
	      #siErrorId := 1;
	      #sbError := True;
	      #sbDone := False;
	      
	      // Wiederholungsauftrag wieder zurücknehmen  
	      #sbWrStart := False;
	      #sbRdStart := False;
	      #sbRead := False;
	      
	      // Fehler : die angeforderte Anzahl Parameter entspricht nicht der übermittelten Anzahl Parameter überein
	    ELSIF NOT (#siParaNo = BYTE_TO_INT(#sxRespParaMulti.sxHeader.syParaNo)) AND NOT #sbRdBusy AND #pbValidSFB THEN
	      #siErrorId := 1;
	      #sbError := True;
	      #sbDone := False;
	      
	      // Wiederholungsauftrag wieder zurücknehmen  
	      #sbWrStart := False;
	      #sbRdStart := False;
	      #sbRead := False;
	      
	      // Fehler : die Achse entspricht nicht der übergebenen Achse
	    ELSIF NOT (#syAxisNo = #sxRespParaMulti.sxHeader.syAxisNo) AND NOT #sbRdBusy AND #pbValidSFB THEN
	      #siErrorId := 1;
	      #sbError := True;
	      #sbDone := False;
	      
	      // Wiederholungsauftrag wieder zurücknehmen  
	      #sbWrStart := False;
	      #sbRdStart := False;
	      #sbRead := False;
	      
	      // kein Fehler beim LESEN AZYKLISCH und Auftrag fertig 
	    ELSIF NOT #sbRdBusy AND #pbValidSFB THEN
	      
	      // die angefragten Parameter auswerten und im Puffer abspeichern
	      #piPointer := 1;
	      #swParaError := 16#0;
	      
	      FOR #piCount := 1 TO #siParaNo DO
	        
	        // ermitteltes Format des Parameters abspeichern
	        #sxParameter[#piCount].syFormat := #sxRespParaMulti.sxData[#piPointer];
	        
	        // Format = Error ? = > gesendeter Parameter fehlerhaft
	        IF (BYTE_TO_INT(#sxRespParaMulti.sxData[#piPointer]) = 68) THEN
	          
	          // Format = Error, zwei Bytes zu übermittelten Fehlernummer zusammenfassen
	          #pwWordHigh := SHL(IN := BYTE_TO_WORD(#sxRespParaMulti.sxData[#piPointer + 2]), N := 8);
	          #pwWordLow := BYTE_TO_WORD(#sxRespParaMulti.sxData[#piPointer + 3]);
	            
	          #sbError := True;
	          
	          // ermittelte Fehlernummer im Puffer abspeichern
	          #sxParameter[#piCount].swErrorNo := #pwWordHigh XOR #pwWordLow;
	          
	          // Die Fehlerhaftigkeit des erkannten Parameter in der Fehlernummer eintragen   
	          IF #piCount = 1 THEN
	            #swParaError := #swParaError OR W#16#01;
	          ELSIF #piCount = 2 THEN
	            #swParaError := #swParaError OR W#16#02;
	          ELSIF #piCount = 3 THEN
	            #swParaError := #swParaError OR W#16#04;
	          ELSIF #piCount = 4 THEN
	            #swParaError := #swParaError OR W#16#08;
	          ELSIF #piCount = 5 THEN
	            #swParaError := #swParaError OR W#16#10;
	          ELSIF #piCount = 6 THEN
	            #swParaError := #swParaError OR W#16#20;
	          ELSIF #piCount = 7 THEN
	            #swParaError := #swParaError OR W#16#40;
	          ELSIF #piCount = 8 THEN
	            #swParaError := #swParaError OR W#16#80;
	          ELSIF #piCount = 9 THEN
	            #swParaError := #swParaError OR W#16#100;
	          ELSIF #piCount = 10 THEN
	            #swParaError := #swParaError OR W#16#200;
	          ELSIF #piCount = 11 THEN
	            #swParaError := #swParaError OR W#16#400;
	          ELSIF #piCount = 12 THEN
	            #swParaError := #swParaError OR W#16#800;
	          ELSIF #piCount = 13 THEN
	            #swParaError := #swParaError OR W#16#1000;
	          ELSIF #piCount = 14 THEN
	            #swParaError := #swParaError OR W#16#2000;
	          ELSIF #piCount = 15 THEN
	            #swParaError := #swParaError OR W#16#4000;
	          ELSIF #piCount = #siParaNo THEN
	            #swParaError := #swParaError OR W#16#8000;
	          END_IF;
	          
	          // Zeiger auf nächsten Parametersatz setzen
	          #piPointer := #piPointer + 6;
	          
	          // Format = Byte ? = > gesendeter Parameter ein Byte lang ohne Vorzeichen
	        ELSIF (#sxRespParaMulti.sxData[#piPointer] = B#16#41) OR (#sxRespParaMulti.sxData[#piPointer] = B#16#05) THEN
	          
	          // ermittelter Parameterwert eintragen (Byte) 
	          #sxParameter[#piCount].srValue := USINT_TO_REAL(BYTE_TO_USINT(#sxRespParaMulti.sxData[#piPointer + 2]));
	          #sxParameter[#piCount].sdValue := 0;
	          
	          // ermittelte Fehlernummer im Puffer zurücksetzen
	          #sxParameter[#piCount].swErrorNo := W#16#00;
	          
	          // Die Fehlerhaftigkeit des erkannten Parameter in der Fehlernummer löschen   
	          IF #piCount = 1 THEN
	            #swParaError := #swParaError AND W#16#FFFE;
	          ELSIF #piCount = 2 THEN
	            #swParaError := #swParaError AND W#16#FFFD;
	          ELSIF #piCount = 3 THEN
	            #swParaError := #swParaError AND W#16#FFFB;
	          ELSIF #piCount = 4 THEN
	            #swParaError := #swParaError AND W#16#FFF7;
	          ELSIF #piCount = 5 THEN
	            #swParaError := #swParaError AND W#16#FFEF;
	          ELSIF #piCount = 6 THEN
	            #swParaError := #swParaError AND W#16#FFDF;
	          ELSIF #piCount = 7 THEN
	            #swParaError := #swParaError AND W#16#FFBF;
	          ELSIF #piCount = 8 THEN
	            #swParaError := #swParaError AND W#16#FF7F;
	          ELSIF #piCount = 9 THEN
	            #swParaError := #swParaError AND W#16#FEFF;
	          ELSIF #piCount = 10 THEN
	            #swParaError := #swParaError AND W#16#FDFF;
	          ELSIF #piCount = 11 THEN
	            #swParaError := #swParaError AND W#16#FBFF;
	          ELSIF #piCount = 12 THEN
	            #swParaError := #swParaError AND W#16#F7FF;
	          ELSIF #piCount = 13 THEN
	            #swParaError := #swParaError AND W#16#EFFF;
	          ELSIF #piCount = 14 THEN
	            #swParaError := #swParaError AND W#16#DFFF;
	          ELSIF #piCount = 15 THEN
	            #swParaError := #swParaError AND W#16#BFFF;
	          ELSIF #piCount = #siParaNo THEN
	            #swParaError := #swParaError AND W#16#7FFF;
	          END_IF;
	          
	          // Zeiger auf nächsten Parametersatz setzen
	          #piPointer := #piPointer + 4;
	          
	          // Format = Byte ? = > gesendeter Parameter ein Byte lang mit Vorzeichen
	        ELSIF (#sxRespParaMulti.sxData[#piPointer] = B#16#02) THEN
	          
	          // ermittelter Parameterwert eintragen (Byte) 
	          #sxParameter[#piCount].srValue := SINT_TO_REAL(BYTE_TO_SINT(#sxRespParaMulti.sxData[#piPointer + 2]));
	          #sxParameter[#piCount].sdValue := 0;
	          
	          // ermittelte Fehlernummer im Puffer zurücksetzen
	          #sxParameter[#piCount].swErrorNo := W#16#00;
	          
	          // Die Fehlerhaftigkeit des erkannten Parameter in der Fehlernummer löschen   
	          IF #piCount = 1 THEN
	            #swParaError := #swParaError AND W#16#FFFE;
	          ELSIF #piCount = 2 THEN
	            #swParaError := #swParaError AND W#16#FFFD;
	          ELSIF #piCount = 3 THEN
	            #swParaError := #swParaError AND W#16#FFFB;
	          ELSIF #piCount = 4 THEN
	            #swParaError := #swParaError AND W#16#FFF7;
	          ELSIF #piCount = 5 THEN
	            #swParaError := #swParaError AND W#16#FFEF;
	          ELSIF #piCount = 6 THEN
	            #swParaError := #swParaError AND W#16#FFDF;
	          ELSIF #piCount = 7 THEN
	            #swParaError := #swParaError AND W#16#FFBF;
	          ELSIF #piCount = 8 THEN
	            #swParaError := #swParaError AND W#16#FF7F;
	          ELSIF #piCount = 9 THEN
	            #swParaError := #swParaError AND W#16#FEFF;
	          ELSIF #piCount = 10 THEN
	            #swParaError := #swParaError AND W#16#FDFF;
	          ELSIF #piCount = 11 THEN
	            #swParaError := #swParaError AND W#16#FBFF;
	          ELSIF #piCount = 12 THEN
	            #swParaError := #swParaError AND W#16#F7FF;
	          ELSIF #piCount = 13 THEN
	            #swParaError := #swParaError AND W#16#EFFF;
	          ELSIF #piCount = 14 THEN
	            #swParaError := #swParaError AND W#16#DFFF;
	          ELSIF #piCount = 15 THEN
	            #swParaError := #swParaError AND W#16#BFFF;
	          ELSIF #piCount = #siParaNo THEN
	            #swParaError := #swParaError AND W#16#7FFF;
	          END_IF;
	          
	          // Zeiger auf nächsten Parametersatz setzen
	          #piPointer := #piPointer + 4;
	          
	          // Format = Word ? = > gesendeter Parameter zwei Bytes lang ohne Vorzeichen
	        ELSIF (#sxRespParaMulti.sxData[#piPointer] = B#16#42) OR (#sxRespParaMulti.sxData[#piPointer] = B#16#06)
	          OR (#sxRespParaMulti.sxData[#piPointer] = B#16#0A) THEN
	          
	          // Format = Word, zwei Bytes zu übermitteltem Parameterwert zusammenfassen
	          #pwWordHigh := SHL(IN := BYTE_TO_WORD(#sxRespParaMulti.sxData[#piPointer + 2]), N := 8);
	          #pwWordLow := BYTE_TO_WORD(#sxRespParaMulti.sxData[#piPointer + 3]);
	          #pwWord1 := #pwWordHigh XOR #pwWordLow;
	          
	          // ermittelter Parameterwert eintragen (Word)
	          #sxParameter[#piCount].srValue := UINT_TO_REAL(WORD_TO_UINT(#pwWord1));
	          #sxParameter[#piCount].sdValue := 0;
	          
	          // ermittelte Fehlernummer im Puffer zurücksetzen
	          #sxParameter[#piCount].swErrorNo := W#16#00;
	          
	          // Die Fehlerhaftigkeit des erkannten Parameter in der Fehlernummer löschen   
	          IF #piCount = 1 THEN
	            #swParaError := #swParaError AND W#16#FFFE;
	          ELSIF #piCount = 2 THEN
	            #swParaError := #swParaError AND W#16#FFFD;
	          ELSIF #piCount = 3 THEN
	            #swParaError := #swParaError AND W#16#FFFB;
	          ELSIF #piCount = 4 THEN
	            #swParaError := #swParaError AND W#16#FFF7;
	          ELSIF #piCount = 5 THEN
	            #swParaError := #swParaError AND W#16#FFEF;
	          ELSIF #piCount = 6 THEN
	            #swParaError := #swParaError AND W#16#FFDF;
	          ELSIF #piCount = 7 THEN
	            #swParaError := #swParaError AND W#16#FFBF;
	          ELSIF #piCount = 8 THEN
	            #swParaError := #swParaError AND W#16#FF7F;
	          ELSIF #piCount = 9 THEN
	            #swParaError := #swParaError AND W#16#FEFF;
	          ELSIF #piCount = 10 THEN
	            #swParaError := #swParaError AND W#16#FDFF;
	          ELSIF #piCount = 11 THEN
	            #swParaError := #swParaError AND W#16#FBFF;
	          ELSIF #piCount = 12 THEN
	            #swParaError := #swParaError AND W#16#F7FF;
	          ELSIF #piCount = 13 THEN
	            #swParaError := #swParaError AND W#16#EFFF;
	          ELSIF #piCount = 14 THEN
	            #swParaError := #swParaError AND W#16#DFFF;
	          ELSIF #piCount = 15 THEN
	            #swParaError := #swParaError AND W#16#BFFF;
	          ELSIF #piCount = #siParaNo THEN
	            #swParaError := #swParaError AND W#16#7FFF;
	          END_IF;
	          
	          // Zeiger auf nächsten Parametersatz setzen
	          #piPointer := #piPointer + 4;
	          
	          // Format = Word ? = > gesendeter Parameter zwei Bytes lang mit Vorzeichen
	        ELSIF (#sxRespParaMulti.sxData[#piPointer] = B#16#03) THEN
	          
	          // Format = Word, zwei Bytes zu übermitteltem Parameterwert zusammenfassen
	          #pwWordHigh := SHL(IN := BYTE_TO_WORD(#sxRespParaMulti.sxData[#piPointer + 2]), N := 8);
	          #pwWordLow := BYTE_TO_WORD(#sxRespParaMulti.sxData[#piPointer + 3]);
	          #pwWord1 := #pwWordHigh XOR #pwWordLow;
	          
	          // ermittelter Parameterwert eintragen (Word)
	          #sxParameter[#piCount].srValue := INT_TO_REAL(WORD_TO_INT(#pwWord1));
	          #sxParameter[#piCount].sdValue := 0;
	          
	          // ermittelte Fehlernummer im Puffer zurücksetzen
	          #sxParameter[#piCount].swErrorNo := W#16#00;
	          
	          // Die Fehlerhaftigkeit des erkannten Parameter in der Fehlernummer löschen   
	          IF #piCount = 1 THEN
	            #swParaError := #swParaError AND W#16#FFFE;
	          ELSIF #piCount = 2 THEN
	            #swParaError := #swParaError AND W#16#FFFD;
	          ELSIF #piCount = 3 THEN
	            #swParaError := #swParaError AND W#16#FFFB;
	          ELSIF #piCount = 4 THEN
	            #swParaError := #swParaError AND W#16#FFF7;
	          ELSIF #piCount = 5 THEN
	            #swParaError := #swParaError AND W#16#FFEF;
	          ELSIF #piCount = 6 THEN
	            #swParaError := #swParaError AND W#16#FFDF;
	          ELSIF #piCount = 7 THEN
	            #swParaError := #swParaError AND W#16#FFBF;
	          ELSIF #piCount = 8 THEN
	            #swParaError := #swParaError AND W#16#FF7F;
	          ELSIF #piCount = 9 THEN
	            #swParaError := #swParaError AND W#16#FEFF;
	          ELSIF #piCount = 10 THEN
	            #swParaError := #swParaError AND W#16#FDFF;
	          ELSIF #piCount = 11 THEN
	            #swParaError := #swParaError AND W#16#FBFF;
	          ELSIF #piCount = 12 THEN
	            #swParaError := #swParaError AND W#16#F7FF;
	          ELSIF #piCount = 13 THEN
	            #swParaError := #swParaError AND W#16#EFFF;
	          ELSIF #piCount = 14 THEN
	            #swParaError := #swParaError AND W#16#DFFF;
	          ELSIF #piCount = 15 THEN
	            #swParaError := #swParaError AND W#16#BFFF;
	          ELSIF #piCount = #siParaNo THEN
	            #swParaError := #swParaError AND W#16#7FFF;
	          END_IF;
	          
	          // Zeiger auf nächsten Parametersatz setzen
	          #piPointer := #piPointer + 4;
	          
	          // Format = Double Word ? = > gesendeter Parameter vier Bytes lang ohne Vorzeichen
	        ELSIF (#sxRespParaMulti.sxData[#piPointer] = B#16#43) OR (#sxRespParaMulti.sxData[#piPointer] = B#16#07) OR
	          (#sxRespParaMulti.sxData[#piPointer] = B#16#0D) THEN
	          
	          // Format = Double Word, vier Bytes zu übermitteltem Parameterwert zusammenfassen
	          #pwWordHigh := SHL(IN := BYTE_TO_WORD(#sxRespParaMulti.sxData[#piPointer + 2]), N := 8);
	          #pwWordLow := BYTE_TO_WORD(#sxRespParaMulti.sxData[#piPointer + 3]);
	          #pwWord1 := #pwWordHigh XOR #pwWordLow;
	          
	          #pwWordHigh := SHL(IN := BYTE_TO_WORD(#sxRespParaMulti.sxData[#piPointer + 4]), N := 8);
	          #pwWordLow := BYTE_TO_WORD(#sxRespParaMulti.sxData[#piPointer + 5]);
	          #pwWord2 := #pwWordHigh XOR #pwWordLow;
	          
	          #pdDWordHigh := SHL(IN := WORD_TO_DWORD(#pwWord1), N := 16);
	          #pdDWordLow := WORD_TO_DWORD(#pwWord2);
	          
	          // ermittelter Parameterwert eintragen (Word)
	          #sxParameter[#piCount].srValue := 0.0;
	          #sxParameter[#piCount].sdValue := DWORD_TO_DINT(#pdDWordHigh XOR #pdDWordLow);
	          
	          // ermittelte Fehlernummer im Puffer zurücksetzen
	          #sxParameter[#piCount].swErrorNo := W#16#00;
	          
	          // Die Fehlerhaftigkeit des erkannten Parameter in der Fehlernummer löschen   
	          IF #piCount = 1 THEN
	            #swParaError := #swParaError AND W#16#FFFE;
	          ELSIF #piCount = 2 THEN
	            #swParaError := #swParaError AND W#16#FFFD;
	          ELSIF #piCount = 3 THEN
	            #swParaError := #swParaError AND W#16#FFFB;
	          ELSIF #piCount = 4 THEN
	            #swParaError := #swParaError AND W#16#FFF7;
	          ELSIF #piCount = 5 THEN
	            #swParaError := #swParaError AND W#16#FFEF;
	          ELSIF #piCount = 6 THEN
	            #swParaError := #swParaError AND W#16#FFDF;
	          ELSIF #piCount = 7 THEN
	            #swParaError := #swParaError AND W#16#FFBF;
	          ELSIF #piCount = 8 THEN
	            #swParaError := #swParaError AND W#16#FF7F;
	          ELSIF #piCount = 9 THEN
	            #swParaError := #swParaError AND W#16#FEFF;
	          ELSIF #piCount = 10 THEN
	            #swParaError := #swParaError AND W#16#FDFF;
	          ELSIF #piCount = 11 THEN
	            #swParaError := #swParaError AND W#16#FBFF;
	          ELSIF #piCount = 12 THEN
	            #swParaError := #swParaError AND W#16#F7FF;
	          ELSIF #piCount = 13 THEN
	            #swParaError := #swParaError AND W#16#EFFF;
	          ELSIF #piCount = 14 THEN
	            #swParaError := #swParaError AND W#16#DFFF;
	          ELSIF #piCount = 15 THEN
	            #swParaError := #swParaError AND W#16#BFFF;
	          ELSIF #piCount = #siParaNo THEN
	            #swParaError := #swParaError AND W#16#7FFF;
	          END_IF;
	          
	          // Zeiger auf nächsten Parametersatz setzen
	          #piPointer := #piPointer + 6;
	          
	          // Format = Double Word ? = > gesendeter Parameter vier Bytes lang mit Vorzeichen
	        ELSIF (#sxRespParaMulti.sxData[#piPointer] = B#16#04) THEN
	          
	          // Format = Double Word, vier Bytes zu übermitteltem Parameterwert zusammenfassen
	          #pwWordHigh := SHL(IN := BYTE_TO_WORD(#sxRespParaMulti.sxData[#piPointer + 2]), N := 8);
	          #pwWordLow := BYTE_TO_WORD(#sxRespParaMulti.sxData[#piPointer + 3]);
	          #pwWord1 := #pwWordHigh XOR #pwWordLow;
	          
	          #pwWordHigh := SHL(IN := BYTE_TO_WORD(#sxRespParaMulti.sxData[#piPointer + 4]), N := 8);
	          #pwWordLow := BYTE_TO_WORD(#sxRespParaMulti.sxData[#piPointer + 5]);
	          #pwWord2 := #pwWordHigh XOR #pwWordLow;
	          
	          #pdDWordHigh := SHL(IN := WORD_TO_DWORD(#pwWord1), N := 16);
	          #pdDWordLow := WORD_TO_DWORD(#pwWord2);
	          
